LIN {X 0,Y 266.128,Z 281.314,A -85,B 0,C 180,E1 -18933.081,E2 -18933.081} C_VEL
LIN {X 0,Y 270.948,Z 292.828,A -85,B 0,C 180,E1 -18934.221,E2 -18934.221} C_VEL
LIN {X 0,Y 268.167,Z 358.472,A -85,B 0,C 180,E1 -18936.067,E2 -18936.067} C_VEL
LIN {X 0,Y 266.983,Z 371.691,A -85,B 0,C 180,E1 -18936.714,E2 -18936.714} C_VEL
LIN {X 0,Y 265.443,Z 384.254,A -85,B 0,C 180,E1 -18937.634,E2 -18937.634} C_VEL
LIN {X 0,Y 263.666,Z 395.639,A -85,B 0,C 180,E1 -18938.771,E2 -18938.771} C_VEL
LIN {X 0,Y 261.611,Z 406.363,A -85,B 0,C 180,E1 -18940.147,E2 -18940.147} C_VEL
LIN {X 0,Y 259.271,Z 416.661,A -85,B 0,C 180,E1 -18941.804,E2 -18941.804} C_VEL
LIN {X 0,Y 257.067,Z 425.49,A -85,B 0,C 180,E1 -18943.574,E2 -18943.574} C_VEL
LIN {X 0,Y 254.605,Z 434.603,A -85,B 0,C 180,E1 -18945.865,E2 -18945.865} C_VEL
LIN {X 0,Y 252.569,Z 441.662,A -85,B 0,C 180,E1 -18948.101,E2 -18948.101} C_VEL
LIN {X 0,Y 250.564,Z 448.509,A -85,B 0,C 180,E1 -18950.869,E2 -18950.869} C_VEL
LIN {X 0,Y 249.045,Z 453.666,A -85,B 0,C 180,E1 -18953.657,E2 -18953.657} C_VEL
LIN {X 0,Y 247.968,Z 457.373,A -85,B 0,C 180,E1 -18956.449,E2 -18956.449} C_VEL
LIN {X 0,Y 247.203,Z 459.794,A -85,B 0,C 180,E1 -18959.22,E2 -18959.22} C_VEL
LIN {X 0,Y 246.741,Z 461.043,A -85,B 0,C 180,E1 -18962.005,E2 -18962.005} C_VEL
LIN {X 0,Y 246.536,Z 461.149,A -85,B 0,C 180,E1 -18964.684,E2 -18964.684} C_VEL
LIN {X 0,Y 246.559,Z 460.631,A -85,B 0,C 180,E1 -18966.48,E2 -18966.48} C_VEL
LIN {X 0,Y 246.666,Z 459.608,A -85,B 0,C 180,E1 -18968.26,E2 -18968.26} C_VEL
LIN {X 0,Y 246.957,Z 458.137,A -85,B 0,C 180,E1 -18970.032,E2 -18970.032} C_VEL
LIN {X 0,Y 247.548,Z 455.004,A -85,B 0,C 180,E1 -18972.656,E2 -18972.656} C_VEL
LIN {X 0,Y 248.257,Z 450.729,A -85,B 0,C 180,E1 -18975.239,E2 -18975.239} C_VEL
LIN {X 0,Y 249.502,Z 444.093,A -85,B 0,C 180,E1 -18978.216,E2 -18978.216} C_VEL
LIN {X 0,Y 250.978,Z 436.828,A -85,B 0,C 180,E1 -18980.734,E2 -18980.734} C_VEL
LIN {X 0,Y 252.458,Z 429.359,A -85,B 0,C 180,E1 -18982.803,E2 -18982.803} C_VEL
LIN {X 0,Y 254.295,Z 419.879,A -85,B 0,C 180,E1 -18984.917,E2 -18984.917} C_VEL
LIN {X 0,Y 256.205,Z 408.995,A -85,B 0,C 180,E1 -18986.855,E2 -18986.855} C_VEL
LIN {X 0,Y 258.11,Z 397.488,A -85,B 0,C 180,E1 -18988.439,E2 -18988.439} C_VEL
LIN {X 0,Y 259.76,Z 384.646,A -85,B 0,C 180,E1 -18989.806,E2 -18989.806} C_VEL
LIN {X 0,Y 261.012,Z 371.674,A -85,B 0,C 180,E1 -18990.807,E2 -18990.807} C_VEL
LIN {X 0,Y 261.936,Z 358.441,A -85,B 0,C 180,E1 -18991.491,E2 -18991.491} C_VEL
LIN {X 0,Y 263.923,Z 304.953,A -85,B 0,C 180,E1 -18993.003,E2 -18993.003} C_VEL
LIN {X 0,Y 264.426,Z 287.5,A -85,B 0,C 180,E1 -18993.493,E2 -18993.493} C_VEL
LIN {X 0,Y 260.391,Z 275.57,A -85,B 0,C 180,E1 -18994.288,E2 -18994.288} C_VEL
LIN {X 0,Y 255.297,Z 263.136,A -85,B 0,C 180,E1 -18995.245,E2 -18995.245} C_VEL
LIN {X 0,Y 249.757,Z 250.129,A -85,B 0,C 180,E1 -18996.361,E2 -18996.361} C_VEL
LIN {X 0,Y 249.402,Z 248.419,A -85,B 0,C 180,E1 -18997.183,E2 -18997.183} C_VEL
LIN {X 0,Y 249.345,Z 248.423,A -85,B 0,C 180,E1 -18999.736,E2 -18999.736} C_VEL
LIN {X 0,Y 249.208,Z 248.445,A -85,B 0,C 180,E1 -19004.703,E2 -19004.703} C_VEL
LIN {X 0,Y 249.142,Z 248.454,A -85,B 0,C 180,E1 -19008.077,E2 -19008.077} C_VEL
LIN {X 0,Y 249.086,Z 248.455,A -85,B 0,C 180,E1 -19011.518,E2 -19011.518} C_VEL
LIN {X 0,Y 249.106,Z 248.455,A -85,B 0,C 180,E1 -19015.469,E2 -19015.469} C_VEL
LIN {X 0,Y 249.04,Z 248.456,A -85,B 0,C 180,E1 -19018.974,E2 -19018.974} C_VEL
LIN {X 0,Y 249.028,Z 248.464,A -85,B 0,C 180,E1 -19022.426,E2 -19022.426} C_VEL
LIN {X 0,Y 249.049,Z 248.456,A -85,B 0,C 180,E1 -19026.341,E2 -19026.341} C_VEL
LIN {X 0,Y 249.006,Z 248.466,A -85,B 0,C 180,E1 -19030.477,E2 -19030.477} C_VEL
LIN {X 0,Y 248.993,Z 248.458,A -85,B 0,C 180,E1 -19034.881,E2 -19034.881} C_VEL
LIN {X 0,Y 249.016,Z 248.463,A -85,B 0,C 180,E1 -19037.362,E2 -19037.362} C_VEL
LIN {X 0,Y 249.044,Z 248.454,A -85,B 0,C 180,E1 -19042.199,E2 -19042.199} C_VEL
LIN {X 0,Y 249.043,Z 248.449,A -85,B 0,C 180,E1 -19045.639,E2 -19045.639} C_VEL
LIN {X 0,Y 249.046,Z 248.46,A -85,B 0,C 180,E1 -19049.472,E2 -19049.472} C_VEL
LIN {X 0,Y 249.071,Z 248.452,A -85,B 0,C 180,E1 -19053.162,E2 -19053.162} C_VEL
LIN {X 0,Y 249.078,Z 248.441,A -85,B 0,C 180,E1 -19056.732,E2 -19056.732} C_VEL
LIN {X 0,Y 249.11,Z 248.452,A -85,B 0,C 180,E1 -19060.211,E2 -19060.211} C_VEL
LIN {X 0,Y 249.241,Z 248.437,A -85,B 0,C 180,E1 -19063.622,E2 -19063.622} C_VEL
LIN {X 0,Y 249.251,Z 248.414,A -85,B 0,C 180,E1 -19068.616,E2 -19068.616} C_VEL
LIN {X 0,Y 249.482,Z 248.398,A -85,B 0,C 180,E1 -19071.903,E2 -19071.903} C_VEL
LIN {X 0,Y 249.435,Z 248.412,A -85,B 0,C 180,E1 -19076.769,E2 -19076.769} C_VEL
LIN {X 0,Y 249.726,Z 248.366,A -85,B 0,C 180,E1 -19080,E2 -19080} C_VEL
LIN {X 0,Y 249.434,Z 248.399,A -85,B 0,C 180,E1 -19083.23,E2 -19083.23} C_VEL
LIN {X 0,Y 249.482,Z 248.409,A -85,B 0,C 180,E1 -19088.097,E2 -19088.097} C_VEL
LIN {X 0,Y 249.251,Z 248.429,A -85,B 0,C 180,E1 -19091.383,E2 -19091.383} C_VEL
LIN {X 0,Y 249.207,Z 248.425,A -85,B 0,C 180,E1 -19092.51,E2 -19092.51} C_VEL
LIN {X 0,Y 248.537,Z 248.51,A -85,B 0,C 180,E1 -19093.859,E2 -19093.859} C_VEL
LIN {X 0,Y 245.637,Z 248.881,A -85,B 0,C 180,E1 -19096.057,E2 -19096.057} C_VEL
LIN {X 0,Y 243.167,Z 249.193,A -85,B 0,C 180,E1 -19097.847,E2 -19097.847} C_VEL
LIN {X 0,Y 242.108,Z 249.325,A -85,B 0,C 180,E1 -19099.238,E2 -19099.238} C_VEL
LIN {X 0,Y 242.022,Z 249.332,A -85,B 0,C 180,E1 -19099.709,E2 -19099.709} C_VEL
LIN {X 0,Y 242.056,Z 249.329,A -85,B 0,C 180,E1 -19103.984,E2 -19103.984} C_VEL
LIN {X 0,Y 242.007,Z 249.336,A -85,B 0,C 180,E1 -19107.687,E2 -19107.687} C_VEL
LIN {X 0,Y 241.973,Z 249.342,A -85,B 0,C 180,E1 -19111.52,E2 -19111.52} C_VEL
LIN {X 0,Y 242.004,Z 249.339,A -85,B 0,C 180,E1 -19115.597,E2 -19115.597} C_VEL
LIN {X 0,Y 241.955,Z 249.345,A -85,B 0,C 180,E1 -19119.719,E2 -19119.719} C_VEL
LIN {X 0,Y 241.922,Z 249.346,A -85,B 0,C 180,E1 -19124.204,E2 -19124.204} C_VEL
LIN {X 0,Y 241.945,Z 249.35,A -85,B 0,C 180,E1 -19128.08,E2 -19128.08} C_VEL
LIN {X 0,Y 242.07,Z 249.446,A -85,B 0,C 180,E1 -19132.786,E2 -19132.786} C_VEL
LIN {X 0,Y 244.245,Z 259.241,A -85,B 0,C 180,E1 -19136.859,E2 -19136.859} C_VEL
LIN {X 0,Y 244.934,Z 262.422,A -85,B 0,C 180,E1 -19138.129,E2 -19138.129} C_VEL
LIN {X 0,Y 252.756,Z 282.367,A -85,B 0,C 180,E1 -19139.716,E2 -19139.716} C_VEL
LIN {X 0,Y 253.632,Z 285.314,A -85,B 0,C 180,E1 -19139.91,E2 -19139.91} C_VEL
LIN {X 0,Y 257.411,Z 312.087,A -85,B 0,C 180,E1 -19141.176,E2 -19141.176} C_VEL
LIN {X 0,Y 255.315,Z 370.97,A -85,B 0,C 180,E1 -19142.877,E2 -19142.877} C_VEL
LIN {X 0,Y 254.099,Z 384.714,A -85,B 0,C 180,E1 -19143.569,E2 -19143.569} C_VEL
LIN {X 0,Y 252.646,Z 397.705,A -85,B 0,C 180,E1 -19144.569,E2 -19144.569} C_VEL
LIN {X 0,Y 250.928,Z 409.521,A -85,B 0,C 180,E1 -19145.82,E2 -19145.82} C_VEL
LIN {X 0,Y 248.993,Z 420.926,A -85,B 0,C 180,E1 -19147.383,E2 -19147.383} C_VEL
LIN {X 0,Y 246.976,Z 431.203,A -85,B 0,C 180,E1 -19149.164,E2 -19149.164} C_VEL
LIN {X 0,Y 245.257,Z 440.449,A -85,B 0,C 180,E1 -19151.192,E2 -19151.192} C_VEL
LIN {X 0,Y 243.708,Z 448.08,A -85,B 0,C 180,E1 -19153.24,E2 -19153.24} C_VEL
LIN {X 0,Y 242.189,Z 455.549,A -85,B 0,C 180,E1 -19155.72,E2 -19155.72} C_VEL
LIN {X 0,Y 241.068,Z 461.533,A -85,B 0,C 180,E1 -19158.225,E2 -19158.225} C_VEL
LIN {X 0,Y 240.366,Z 466.244,A -85,B 0,C 180,E1 -19160.746,E2 -19160.746} C_VEL
LIN {X 0,Y 239.953,Z 469.818,A -85,B 0,C 180,E1 -19163.272,E2 -19163.272} C_VEL
LIN {X 0,Y 239.797,Z 471.831,A -85,B 0,C 180,E1 -19165.189,E2 -19165.189} C_VEL
LIN {X 0,Y 239.84,Z 473.941,A -85,B 0,C 180,E1 -19168.321,E2 -19168.321} C_VEL
LIN {X 0,Y 239.913,Z 474.499,A -85,B 0,C 180,E1 -19170,E2 -19170} C_VEL
LIN {X 0,Y 239.83,Z 474.623,A -85,B 0,C 180,E1 -19171.679,E2 -19171.679} C_VEL
LIN {X 0,Y 239.801,Z 473.657,A -85,B 0,C 180,E1 -19175.044,E2 -19175.044} C_VEL
LIN {X 0,Y 239.952,Z 472.594,A -85,B 0,C 180,E1 -19176.728,E2 -19176.728} C_VEL
LIN {X 0,Y 240.217,Z 471.104,A -85,B 0,C 180,E1 -19178.412,E2 -19178.412} C_VEL
LIN {X 0,Y 240.899,Z 468.07,A -85,B 0,C 180,E1 -19180.931,E2 -19180.931} C_VEL
LIN {X 0,Y 241.929,Z 463.995,A -85,B 0,C 180,E1 -19183.439,E2 -19183.439} C_VEL
LIN {X 0,Y 243.832,Z 457.761,A -85,B 0,C 180,E1 -19186.322,E2 -19186.322} C_VEL
LIN {X 0,Y 245.809,Z 450.997,A -85,B 0,C 180,E1 -19188.763,E2 -19188.763} C_VEL
LIN {X 0,Y 248.119,Z 442.786,A -85,B 0,C 180,E1 -19191.127,E2 -19191.127} C_VEL
LIN {X 0,Y 250.503,Z 434.045,A -85,B 0,C 180,E1 -19193.128,E2 -19193.128} C_VEL
LIN {X 0,Y 253.281,Z 423.502,A -85,B 0,C 180,E1 -19195.034,E2 -19195.034} C_VEL
LIN {X 0,Y 255.661,Z 413.101,A -85,B 0,C 180,E1 -19196.532,E2 -19196.532} C_VEL
LIN {X 0,Y 257.925,Z 401.697,A -85,B 0,C 180,E1 -19197.816,E2 -19197.816} C_VEL
LIN {X 0,Y 259.929,Z 388.71,A -85,B 0,C 180,E1 -19198.902,E2 -19198.902} C_VEL
LIN {X 0,Y 261.485,Z 375.958,A -85,B 0,C 180,E1 -19199.637,E2 -19199.637} C_VEL
LIN {X 0,Y 262.379,Z 362.672,A -85,B 0,C 180,E1 -19200.122,E2 -19200.122} C_VEL
LIN {X 0,Y 264.36,Z 313.239,A -85,B 0,C 180,E1 -19201.529,E2 -19201.529} C_VEL
LIN {X 0,Y 261.649,Z 294.723,A -85,B 0,C 180,E1 -19202.614,E2 -19202.614} C_VEL
LIN {X 0,Y 257.644,Z 285.16,A -85,B 0,C 180,E1 -19203.642,E2 -19203.642} C_VEL
LIN {X 0,Y 251.833,Z 273.124,A -85,B 0,C 180,E1 -19205.159,E2 -19205.159} C_VEL
LIN {X 0,Y 247.323,Z 264.812,A -85,B 0,C 180,E1 -19206.38,E2 -19206.38} C_VEL
LIN {X 0,Y 245.234,Z 260.708,A -85,B 0,C 180,E1 -19207.001,E2 -19207.001} C_VEL
LIN {X 0,Y 243.213,Z 253.602,A -85,B 0,C 180,E1 -19210.512,E2 -19210.512} C_VEL
LIN {X 0,Y 241.96,Z 249.343,A -85,B 0,C 180,E1 -19212.873,E2 -19212.873} C_VEL
LIN {X 0,Y 241.932,Z 249.352,A -85,B 0,C 180,E1 -19216.572,E2 -19216.572} C_VEL
LIN {X 0,Y 241.957,Z 249.345,A -85,B 0,C 180,E1 -19220.281,E2 -19220.281} C_VEL
LIN {X 0,Y 241.988,Z 249.334,A -85,B 0,C 180,E1 -19224.489,E2 -19224.489} C_VEL
LIN {X 0,Y 241.974,Z 249.333,A -85,B 0,C 180,E1 -19228.48,E2 -19228.48} C_VEL
LIN {X 0,Y 242.008,Z 249.329,A -85,B 0,C 180,E1 -19232.313,E2 -19232.313} C_VEL
LIN {X 0,Y 242.058,Z 249.326,A -85,B 0,C 180,E1 -19236.016,E2 -19236.016} C_VEL
LIN {X 0,Y 242.038,Z 249.335,A -85,B 0,C 180,E1 -19239.608,E2 -19239.608} C_VEL
LIN {X 0,Y 242.164,Z 249.32,A -85,B 0,C 180,E1 -19243.278,E2 -19243.278} C_VEL
LIN {X 0,Y 242.187,Z 249.316,A -85,B 0,C 180,E1 -19248.28,E2 -19248.28} C_VEL
LIN {X 0,Y 242.427,Z 249.28,A -85,B 0,C 180,E1 -19251.666,E2 -19251.666} C_VEL
LIN {X 0,Y 242.258,Z 249.296,A -85,B 0,C 180,E1 -19255.007,E2 -19255.007} C_VEL
LIN {X 0,Y 242.636,Z 249.257,A -85,B 0,C 180,E1 -19258.34,E2 -19258.34} C_VEL
LIN {X 0,Y 242.636,Z 249.261,A -85,B 0,C 180,E1 -19261.66,E2 -19261.66} C_VEL
LIN {X 0,Y 242.43,Z 249.284,A -85,B 0,C 180,E1 -19266.708,E2 -19266.708} C_VEL
LIN {X 0,Y 242.315,Z 249.302,A -85,B 0,C 180,E1 -19270.022,E2 -19270.022} C_VEL
LIN {X 0,Y 242.168,Z 249.313,A -85,B 0,C 180,E1 -19275.141,E2 -19275.141} C_VEL
LIN {X 0,Y 242.073,Z 249.326,A -85,B 0,C 180,E1 -19278.624,E2 -19278.624} C_VEL
LIN {X 0,Y 242.006,Z 249.34,A -85,B 0,C 180,E1 -19282.181,E2 -19282.181} C_VEL
LIN {X 0,Y 242.035,Z 249.495,A -85,B 0,C 180,E1 -19286.516,E2 -19286.516} C_VEL
LIN {X 0,Y 242.596,Z 251.41,A -85,B 0,C 180,E1 -19287.498,E2 -19287.498} C_VEL
LIN {X 0,Y 245.302,Z 255.739,A -85,B 0,C 180,E1 -19288.27,E2 -19288.27} C_VEL
LIN {X 0,Y 252.844,Z 268.592,A -85,B 0,C 180,E1 -19290.302,E2 -19290.302} C_VEL
LIN {X 0,Y 259.452,Z 281.589,A -85,B 0,C 180,E1 -19291.986,E2 -19291.986} C_VEL
LIN {X 0,Y 265.197,Z 295.065,A -85,B 0,C 180,E1 -19293.413,E2 -19293.413} C_VEL
LIN {X 0,Y 262.301,Z 358.088,A -85,B 0,C 180,E1 -19295.194,E2 -19295.194} C_VEL
LIN {X 0,Y 261.078,Z 371.499,A -85,B 0,C 180,E1 -19295.854,E2 -19295.854} C_VEL
LIN {X 0,Y 259.42,Z 384.584,A -85,B 0,C 180,E1 -19296.826,E2 -19296.826} C_VEL
LIN {X 0,Y 257.557,Z 395.918,A -85,B 0,C 180,E1 -19297.983,E2 -19297.983} C_VEL
LIN {X 0,Y 255.153,Z 407.642,A -85,B 0,C 180,E1 -19299.535,E2 -19299.535} C_VEL
LIN {X 0,Y 252.626,Z 418.187,A -85,B 0,C 180,E1 -19301.311,E2 -19301.311} C_VEL
LIN {X 0,Y 250.347,Z 426.756,A -85,B 0,C 180,E1 -19303.122,E2 -19303.122} C_VEL
LIN {X 0,Y 247.771,Z 435.677,A -85,B 0,C 180,E1 -19305.482,E2 -19305.482} C_VEL
LIN {X 0,Y 245.384,Z 443.543,A -85,B 0,C 180,E1 -19308.131,E2 -19308.131} C_VEL
LIN {X 0,Y 243.614,Z 449.235,A -85,B 0,C 180,E1 -19310.604,E2 -19310.604} C_VEL
LIN {X 0,Y 242.015,Z 454.238,A -85,B 0,C 180,E1 -19313.465,E2 -19313.465} C_VEL
LIN {X 0,Y 240.912,Z 457.841,A -85,B 0,C 180,E1 -19316.339,E2 -19316.339} C_VEL
LIN {X 0,Y 240.328,Z 459.538,A -85,B 0,C 180,E1 -19318.239,E2 -19318.239} C_VEL
LIN {X 0,Y 239.678,Z 461.188,A -85,B 0,C 180,E1 -19321.605,E2 -19321.605} C_VEL
LIN {X 0,Y 239.472,Z 461.423,A -85,B 0,C 180,E1 -19323.882,E2 -19323.882} C_VEL
LIN {X 0,Y 239.47,Z 461.061,A -85,B 0,C 180,E1 -19325.74,E2 -19325.74} C_VEL
LIN {X 0,Y 239.5,Z 460.259,A -85,B 0,C 180,E1 -19327.575,E2 -19327.575} C_VEL
LIN {X 0,Y 239.781,Z 458.661,A -85,B 0,C 180,E1 -19329.707,E2 -19329.707} C_VEL
LIN {X 0,Y 240.32,Z 456.053,A -85,B 0,C 180,E1 -19332.117,E2 -19332.117} C_VEL
LIN {X 0,Y 241.024,Z 452.063,A -85,B 0,C 180,E1 -19334.786,E2 -19334.786} C_VEL
LIN {X 0,Y 242,Z 446.849,A -85,B 0,C 180,E1 -19337.419,E2 -19337.419} C_VEL
LIN {X 0,Y 243.365,Z 440.237,A -85,B 0,C 180,E1 -19340.022,E2 -19340.022} C_VEL
LIN {X 0,Y 245.116,Z 431.875,A -85,B 0,C 180,E1 -19342.587,E2 -19342.587} C_VEL
LIN {X 0,Y 246.993,Z 422.758,A -85,B 0,C 180,E1 -19344.813,E2 -19344.813} C_VEL
LIN {X 0,Y 248.864,Z 412.772,A -85,B 0,C 180,E1 -19346.762,E2 -19346.762} C_VEL
LIN {X 0,Y 250.734,Z 402.199,A -85,B 0,C 180,E1 -19348.394,E2 -19348.394} C_VEL
LIN {X 0,Y 252.416,Z 390.682,A -85,B 0,C 180,E1 -19349.8,E2 -19349.8} C_VEL
LIN {X 0,Y 253.89,Z 378.372,A -85,B 0,C 180,E1 -19350.94,E2 -19350.94} C_VEL
LIN {X 0,Y 254.975,Z 365.675,A -85,B 0,C 180,E1 -19351.775,E2 -19351.775} C_VEL
LIN {X 0,Y 255.729,Z 352.726,A -85,B 0,C 180,E1 -19352.317,E2 -19352.317} C_VEL
LIN {X 0,Y 257.984,Z 288.658,A -85,B 0,C 180,E1 -19354.129,E2 -19354.129} C_VEL
LIN {X 0,Y 251.527,Z 270.992,A -85,B 0,C 180,E1 -19355.416,E2 -19355.416} C_VEL
LIN {X 0,Y 242.616,Z 250.421,A -85,B 0,C 180,E1 -19357.202,E2 -19357.202} C_VEL
LIN {X 0,Y 242.383,Z 249.294,A -85,B 0,C 180,E1 -19357.706,E2 -19357.706} C_VEL
LIN {X 0,Y 242.182,Z 249.319,A -85,B 0,C 180,E1 -19361.72,E2 -19361.72} C_VEL
LIN {X 0,Y 242.165,Z 249.323,A -85,B 0,C 180,E1 -19366.721,E2 -19366.721} C_VEL
LIN {X 0,Y 242.027,Z 249.332,A -85,B 0,C 180,E1 -19371.686,E2 -19371.686} C_VEL
LIN {X 0,Y 242.033,Z 249.338,A -85,B 0,C 180,E1 -19375.82,E2 -19375.82} C_VEL
LIN {X 0,Y 241.97,Z 249.338,A -85,B 0,C 180,E1 -19379.588,E2 -19379.588} C_VEL
LIN {X 0,Y 241.98,Z 249.343,A -85,B 0,C 180,E1 -19383.492,E2 -19383.492} C_VEL
LIN {X 0,Y 241.99,Z 249.337,A -85,B 0,C 180,E1 -19387.581,E2 -19387.581} C_VEL
LIN {X 0,Y 241.933,Z 249.343,A -85,B 0,C 180,E1 -19391.923,E2 -19391.923} C_VEL
LIN {X 0,Y 241.932,Z 249.345,A -85,B 0,C 180,E1 -19396.571,E2 -19396.571} C_VEL
LIN {X 0,Y 241.956,Z 249.343,A -85,B 0,C 180,E1 -19400.28,E2 -19400.28} C_VEL
LIN {X 0,Y 241.987,Z 249.324,A -85,B 0,C 180,E1 -19404.489,E2 -19404.489} C_VEL
LIN {X 0,Y 241.972,Z 249.342,A -85,B 0,C 180,E1 -19408.479,E2 -19408.479} C_VEL
LIN {X 0,Y 242.002,Z 249.334,A -85,B 0,C 180,E1 -19412.312,E2 -19412.312} C_VEL
LIN {X 0,Y 242.056,Z 249.312,A -85,B 0,C 180,E1 -19416.016,E2 -19416.016} C_VEL
LIN {X 0,Y 242.036,Z 249.328,A -85,B 0,C 180,E1 -19419.608,E2 -19419.608} C_VEL
LIN {X 0,Y 242.162,Z 249.318,A -85,B 0,C 180,E1 -19423.278,E2 -19423.278} C_VEL
LIN {X 0,Y 242.185,Z 249.294,A -85,B 0,C 180,E1 -19428.28,E2 -19428.28} C_VEL
LIN {X 0,Y 242.433,Z 249.274,A -85,B 0,C 180,E1 -19431.666,E2 -19431.666} C_VEL
LIN {X 0,Y 242.259,Z 249.306,A -85,B 0,C 180,E1 -19435.007,E2 -19435.007} C_VEL
LIN {X 0,Y 242.635,Z 249.255,A -85,B 0,C 180,E1 -19438.34,E2 -19438.34} C_VEL
LIN {X 0,Y 242.634,Z 249.241,A -85,B 0,C 180,E1 -19441.66,E2 -19441.66} C_VEL
LIN {X 0,Y 242.432,Z 249.286,A -85,B 0,C 180,E1 -19446.659,E2 -19446.659} C_VEL
LIN {X 0,Y 242.344,Z 249.296,A -85,B 0,C 180,E1 -19450.02,E2 -19450.02} C_VEL
LIN {X 0,Y 242.165,Z 249.31,A -85,B 0,C 180,E1 -19455.141,E2 -19455.141} C_VEL
LIN {X 0,Y 242.072,Z 249.331,A -85,B 0,C 180,E1 -19458.624,E2 -19458.624} C_VEL
LIN {X 0,Y 242.022,Z 249.332,A -85,B 0,C 180,E1 -19459.709,E2 -19459.709} C_VEL
LIN {X 0,Y 241.363,Z 249.417,A -85,B 0,C 180,E1 -19461.098,E2 -19461.098} C_VEL
LIN {X 0,Y 238.532,Z 249.775,A -85,B 0,C 180,E1 -19463.364,E2 -19463.364} C_VEL
LIN {X 0,Y 236.107,Z 250.077,A -85,B 0,C 180,E1 -19465.209,E2 -19465.209} C_VEL
LIN {X 0,Y 235.04,Z 250.206,A -85,B 0,C 180,E1 -19466.641,E2 -19466.641} C_VEL
LIN {X 0,Y 234.939,Z 250.214,A -85,B 0,C 180,E1 -19467.127,E2 -19467.127} C_VEL
LIN {X 0,Y 234.93,Z 250.222,A -85,B 0,C 180,E1 -19470.568,E2 -19470.568} C_VEL
LIN {X 0,Y 234.929,Z 250.221,A -85,B 0,C 180,E1 -19474.638,E2 -19474.638} C_VEL
LIN {X 0,Y 234.94,Z 250.219,A -85,B 0,C 180,E1 -19478.945,E2 -19478.945} C_VEL
LIN {X 0,Y 234.879,Z 250.219,A -85,B 0,C 180,E1 -19483.488,E2 -19483.488} C_VEL
LIN {X 0,Y 234.886,Z 250.227,A -85,B 0,C 180,E1 -19486.514,E2 -19486.514} C_VEL
LIN {X 0,Y 234.954,Z 250.212,A -85,B 0,C 180,E1 -19491.086,E2 -19491.086} C_VEL
LIN {X 0,Y 235.002,Z 250.334,A -85,B 0,C 180,E1 -19492.121,E2 -19492.121} C_VEL
LIN {X 0,Y 237.1,Z 259.527,A -85,B 0,C 180,E1 -19496.095,E2 -19496.095} C_VEL
LIN {X 0,Y 237.716,Z 262.328,A -85,B 0,C 180,E1 -19497.215,E2 -19497.215} C_VEL
LIN {X 0,Y 245.795,Z 282.465,A -85,B 0,C 180,E1 -19498.919,E2 -19498.919} C_VEL
LIN {X 0,Y 247.395,Z 287.334,A -85,B 0,C 180,E1 -19499.272,E2 -19499.272} C_VEL
LIN {X 0,Y 250.943,Z 313.525,A -85,B 0,C 180,E1 -19500.542,E2 -19500.542} C_VEL
LIN {X 0,Y 248.759,Z 371.621,A -85,B 0,C 180,E1 -19502.272,E2 -19502.272} C_VEL
LIN {X 0,Y 247.494,Z 385.083,A -85,B 0,C 180,E1 -19502.978,E2 -19502.978} C_VEL
LIN {X 0,Y 246.095,Z 397.387,A -85,B 0,C 180,E1 -19503.955,E2 -19503.955} C_VEL
LIN {X 0,Y 244.453,Z 408.44,A -85,B 0,C 180,E1 -19505.136,E2 -19505.136} C_VEL
LIN {X 0,Y 242.432,Z 420.007,A -85,B 0,C 180,E1 -19506.736,E2 -19506.736} C_VEL
LIN {X 0,Y 240.331,Z 430.432,A -85,B 0,C 180,E1 -19508.56,E2 -19508.56} C_VEL
LIN {X 0,Y 238.299,Z 440.691,A -85,B 0,C 180,E1 -19510.863,E2 -19510.863} C_VEL
LIN {X 0,Y 236.893,Z 447.513,A -85,B 0,C 180,E1 -19512.742,E2 -19512.742} C_VEL
LIN {X 0,Y 235.295,Z 455.05,A -85,B 0,C 180,E1 -19515.293,E2 -19515.293} C_VEL
LIN {X 0,Y 234.061,Z 461.09,A -85,B 0,C 180,E1 -19517.867,E2 -19517.867} C_VEL
LIN {X 0,Y 233.314,Z 465.856,A -85,B 0,C 180,E1 -19520.464,E2 -19520.464} C_VEL
LIN {X 0,Y 232.888,Z 469.48,A -85,B 0,C 180,E1 -19523.067,E2 -19523.067} C_VEL
LIN {X 0,Y 232.715,Z 471.736,A -85,B 0,C 180,E1 -19525.277,E2 -19525.277} C_VEL
LIN {X 0,Y 232.752,Z 473.691,A -85,B 0,C 180,E1 -19528.27,E2 -19528.27} C_VEL
LIN {X 0,Y 232.822,Z 474.269,A -85,B 0,C 180,E1 -19530,E2 -19530} C_VEL
LIN {X 0,Y 232.742,Z 474.435,A -85,B 0,C 180,E1 -19531.731,E2 -19531.731} C_VEL
LIN {X 0,Y 232.731,Z 473.513,A -85,B 0,C 180,E1 -19535.198,E2 -19535.198} C_VEL
LIN {X 0,Y 232.89,Z 472.471,A -85,B 0,C 180,E1 -19536.933,E2 -19536.933} C_VEL
LIN {X 0,Y 233.186,Z 471.023,A -85,B 0,C 180,E1 -19538.667,E2 -19538.667} C_VEL
LIN {X 0,Y 233.914,Z 468.025,A -85,B 0,C 180,E1 -19541.262,E2 -19541.262} C_VEL
LIN {X 0,Y 234.997,Z 463.995,A -85,B 0,C 180,E1 -19543.843,E2 -19543.843} C_VEL
LIN {X 0,Y 237.028,Z 457.826,A -85,B 0,C 180,E1 -19546.804,E2 -19546.804} C_VEL
LIN {X 0,Y 239.431,Z 450.096,A -85,B 0,C 180,E1 -19549.656,E2 -19549.656} C_VEL
LIN {X 0,Y 241.509,Z 443.011,A -85,B 0,C 180,E1 -19551.734,E2 -19551.734} C_VEL
LIN {X 0,Y 244.01,Z 434.411,A -85,B 0,C 180,E1 -19553.78,E2 -19553.78} C_VEL
LIN {X 0,Y 246.902,Z 423.998,A -85,B 0,C 180,E1 -19555.727,E2 -19555.727} C_VEL
LIN {X 0,Y 249.372,Z 413.743,A -85,B 0,C 180,E1 -19557.256,E2 -19557.256} C_VEL
LIN {X 0,Y 251.714,Z 402.56,A -85,B 0,C 180,E1 -19558.564,E2 -19558.564} C_VEL
LIN {X 0,Y 253.793,Z 390.029,A -85,B 0,C 180,E1 -19559.669,E2 -19559.669} C_VEL
LIN {X 0,Y 255.483,Z 376.775,A -85,B 0,C 180,E1 -19560.477,E2 -19560.477} C_VEL
LIN {X 0,Y 256.48,Z 363.996,A -85,B 0,C 180,E1 -19560.973,E2 -19560.973} C_VEL
LIN {X 0,Y 258.585,Z 314.433,A -85,B 0,C 180,E1 -19562.41,E2 -19562.41} C_VEL
LIN {X 0,Y 256.155,Z 297.133,A -85,B 0,C 180,E1 -19563.459,E2 -19563.459} C_VEL
LIN {X 0,Y 249.704,Z 282.43,A -85,B 0,C 180,E1 -19565.205,E2 -19565.205} C_VEL
LIN {X 0,Y 243.232,Z 269.908,A -85,B 0,C 180,E1 -19567.029,E2 -19567.029} C_VEL
LIN {X 0,Y 239.919,Z 264.16,A -85,B 0,C 180,E1 -19568.002,E2 -19568.002} C_VEL
LIN {X 0,Y 237.878,Z 260.328,A -85,B 0,C 180,E1 -19568.689,E2 -19568.689} C_VEL
LIN {X 0,Y 235.649,Z 252.613,A -85,B 0,C 180,E1 -19572.815,E2 -19572.815} C_VEL
LIN {X 0,Y 234.88,Z 250.228,A -85,B 0,C 180,E1 -19574.224,E2 -19574.224} C_VEL
LIN {X 0,Y 234.883,Z 250.223,A -85,B 0,C 180,E1 -19578.832,E2 -19578.832} C_VEL
LIN {X 0,Y 234.918,Z 250.216,A -85,B 0,C 180,E1 -19581.079,E2 -19581.079} C_VEL
LIN {X 0,Y 234.931,Z 250.212,A -85,B 0,C 180,E1 -19585.362,E2 -19585.362} C_VEL
LIN {X 0,Y 234.932,Z 250.212,A -85,B 0,C 180,E1 -19589.432,E2 -19589.432} C_VEL
LIN {X 0,Y 234.995,Z 250.207,A -85,B 0,C 180,E1 -19593.794,E2 -19593.794} C_VEL
LIN {X 0,Y 235.012,Z 250.212,A -85,B 0,C 180,E1 -19598.97,E2 -19598.97} C_VEL
LIN {X 0,Y 235.097,Z 250.197,A -85,B 0,C 180,E1 -19603.059,E2 -19603.059} C_VEL
LIN {X 0,Y 235.147,Z 250.193,A -85,B 0,C 180,E1 -19607.924,E2 -19607.924} C_VEL
LIN {X 0,Y 235.376,Z 250.155,A -85,B 0,C 180,E1 -19611.414,E2 -19611.414} C_VEL
LIN {X 0,Y 235.403,Z 250.161,A -85,B 0,C 180,E1 -19613.141,E2 -19613.141} C_VEL
LIN {X 0,Y 235.596,Z 250.134,A -85,B 0,C 180,E1 -19618.291,E2 -19618.291} C_VEL
LIN {X 0,Y 235.596,Z 250.138,A -85,B 0,C 180,E1 -19621.71,E2 -19621.71} C_VEL
LIN {X 0,Y 235.404,Z 250.158,A -85,B 0,C 180,E1 -19626.859,E2 -19626.859} C_VEL
LIN {X 0,Y 235.239,Z 250.183,A -85,B 0,C 180,E1 -19630.327,E2 -19630.327} C_VEL
LIN {X 0,Y 235.115,Z 250.192,A -85,B 0,C 180,E1 -19635.607,E2 -19635.607} C_VEL
LIN {X 0,Y 235.009,Z 250.209,A -85,B 0,C 180,E1 -19639.206,E2 -19639.206} C_VEL
LIN {X 0,Y 234.951,Z 250.219,A -85,B 0,C 180,E1 -19642.884,E2 -19642.884} C_VEL
LIN {X 0,Y 234.981,Z 250.31,A -85,B 0,C 180,E1 -19645.071,E2 -19645.071} C_VEL
LIN {X 0,Y 235.378,Z 251.736,A -85,B 0,C 180,E1 -19645.82,E2 -19645.82} C_VEL
LIN {X 0,Y 237.58,Z 255.347,A -85,B 0,C 180,E1 -19646.519,E2 -19646.519} C_VEL
LIN {X 0,Y 239.548,Z 258.341,A -85,B 0,C 180,E1 -19647.108,E2 -19647.108} C_VEL
LIN {X 0,Y 246.236,Z 269.361,A -85,B 0,C 180,E1 -19649.026,E2 -19649.026} C_VEL
LIN {X 0,Y 253.083,Z 282.429,A -85,B 0,C 180,E1 -19650.877,E2 -19650.877} C_VEL
LIN {X 0,Y 259.209,Z 296.474,A -85,B 0,C 180,E1 -19652.49,E2 -19652.49} C_VEL
LIN {X 0,Y 259.342,Z 298.411,A -85,B 0,C 180,E1 -19652.583,E2 -19652.583} C_VEL
LIN {X 0,Y 256.343,Z 359.418,A -85,B 0,C 180,E1 -19654.35,E2 -19654.35} C_VEL
LIN {X 0,Y 255.027,Z 373.007,A -85,B 0,C 180,E1 -19655.057,E2 -19655.057} C_VEL
LIN {X 0,Y 253.367,Z 385.354,A -85,B 0,C 180,E1 -19656.017,E2 -19656.017} C_VEL
LIN {X 0,Y 251.426,Z 396.504,A -85,B 0,C 180,E1 -19657.189,E2 -19657.189} C_VEL
LIN {X 0,Y 248.958,Z 408.041,A -85,B 0,C 180,E1 -19658.754,E2 -19658.754} C_VEL
LIN {X 0,Y 246.251,Z 418.766,A -85,B 0,C 180,E1 -19660.608,E2 -19660.608} C_VEL
LIN {X 0,Y 243.636,Z 428.009,A -85,B 0,C 180,E1 -19662.644,E2 -19662.644} C_VEL
LIN {X 0,Y 240.979,Z 436.765,A -85,B 0,C 180,E1 -19665.074,E2 -19665.074} C_VEL
LIN {X 0,Y 238.811,Z 443.431,A -85,B 0,C 180,E1 -19667.401,E2 -19667.401} C_VEL
LIN {X 0,Y 236.833,Z 449.403,A -85,B 0,C 180,E1 -19670.045,E2 -19670.045} C_VEL
LIN {X 0,Y 235.454,Z 453.353,A -85,B 0,C 180,E1 -19672.273,E2 -19672.273} C_VEL
LIN {X 0,Y 234.173,Z 457.304,A -85,B 0,C 180,E1 -19675.234,E2 -19675.234} C_VEL
LIN {X 0,Y 233.451,Z 459.372,A -85,B 0,C 180,E1 -19677.452,E2 -19677.452} C_VEL
LIN {X 0,Y 232.993,Z 460.521,A -85,B 0,C 180,E1 -19679.15,E2 -19679.15} C_VEL
LIN {X 0,Y 232.644,Z 461.333,A -85,B 0,C 180,E1 -19681.172,E2 -19681.172} C_VEL
LIN {X 0,Y 232.426,Z 461.63,A -85,B 0,C 180,E1 -19683.027,E2 -19683.027} C_VEL
LIN {X 0,Y 232.352,Z 461.404,A -85,B 0,C 180,E1 -19685.152,E2 -19685.152} C_VEL
LIN {X 0,Y 232.363,Z 460.788,A -85,B 0,C 180,E1 -19686.846,E2 -19686.846} C_VEL
LIN {X 0,Y 232.672,Z 459.096,A -85,B 0,C 180,E1 -19689.452,E2 -19689.452} C_VEL
LIN {X 0,Y 233.305,Z 455.934,A -85,B 0,C 180,E1 -19692.468,E2 -19692.468} C_VEL
LIN {X 0,Y 234.039,Z 451.844,A -85,B 0,C 180,E1 -19695.212,E2 -19695.212} C_VEL
LIN {X 0,Y 235.099,Z 446.516,A -85,B 0,C 180,E1 -19697.921,E2 -19697.921} C_VEL
LIN {X 0,Y 236.564,Z 439.723,A -85,B 0,C 180,E1 -19700.596,E2 -19700.596} C_VEL
LIN {X 0,Y 238.424,Z 431.205,A -85,B 0,C 180,E1 -19703.228,E2 -19703.228} C_VEL
LIN {X 0,Y 240.291,Z 422.458,A -85,B 0,C 180,E1 -19705.386,E2 -19705.386} C_VEL
LIN {X 0,Y 242.145,Z 412.834,A -85,B 0,C 180,E1 -19707.296,E2 -19707.296} C_VEL
LIN {X 0,Y 244.085,Z 402.231,A -85,B 0,C 180,E1 -19708.969,E2 -19708.969} C_VEL
LIN {X 0,Y 245.83,Z 390.664,A -85,B 0,C 180,E1 -19710.411,E2 -19710.411} C_VEL
LIN {X 0,Y 247.236,Z 379.371,A -85,B 0,C 180,E1 -19711.489,E2 -19711.489} C_VEL
LIN {X 0,Y 248.361,Z 367.271,A -85,B 0,C 180,E1 -19712.331,E2 -19712.331} C_VEL
LIN {X 0,Y 249.157,Z 353.963,A -85,B 0,C 180,E1 -19712.93,E2 -19712.93} C_VEL
LIN {X 0,Y 251.626,Z 290.598,A -85,B 0,C 180,E1 -19714.755,E2 -19714.755} C_VEL
LIN {X 0,Y 245.646,Z 274.036,A -85,B 0,C 180,E1 -19716.004,E2 -19716.004} C_VEL
LIN {X 0,Y 236.224,Z 252.784,A -85,B 0,C 180,E1 -19717.934,E2 -19717.934} C_VEL
LIN {X 0,Y 235.433,Z 250.591,A -85,B 0,C 180,E1 -19718.152,E2 -19718.152} C_VEL
LIN {X 0,Y 235.338,Z 250.174,A -85,B 0,C 180,E1 -19718.371,E2 -19718.371} C_VEL
LIN {X 0,Y 235.116,Z 250.199,A -85,B 0,C 180,E1 -19722.078,E2 -19722.078} C_VEL
LIN {X 0,Y 235.099,Z 250.204,A -85,B 0,C 180,E1 -19726.94,E2 -19726.94} C_VEL
LIN {X 0,Y 234.99,Z 250.205,A -85,B 0,C 180,E1 -19732.006,E2 -19732.006} C_VEL
LIN {X 0,Y 234.947,Z 250.216,A -85,B 0,C 180,E1 -19736.66,E2 -19736.66} C_VEL
LIN {X 0,Y 234.9,Z 250.224,A -85,B 0,C 180,E1 -19740.572,E2 -19740.572} C_VEL
LIN {X 0,Y 234.931,Z 250.212,A -85,B 0,C 180,E1 -19744.637,E2 -19744.637} C_VEL
LIN {X 0,Y 234.942,Z 250.218,A -85,B 0,C 180,E1 -19748.944,E2 -19748.944} C_VEL
LIN {X 0,Y 234.88,Z 250.215,A -85,B 0,C 180,E1 -19753.487,E2 -19753.487} C_VEL
LIN {X 0,Y 234.885,Z 250.223,A -85,B 0,C 180,E1 -19756.513,E2 -19756.513} C_VEL
LIN {X 0,Y 234.918,Z 250.218,A -85,B 0,C 180,E1 -19761.078,E2 -19761.078} C_VEL
LIN {X 0,Y 234.93,Z 250.203,A -85,B 0,C 180,E1 -19765.362,E2 -19765.362} C_VEL
LIN {X 0,Y 234.921,Z 250.22,A -85,B 0,C 180,E1 -19769.43,E2 -19769.43} C_VEL
LIN {X 0,Y 234.993,Z 250.201,A -85,B 0,C 180,E1 -19773.794,E2 -19773.794} C_VEL
LIN {X 0,Y 235.01,Z 250.202,A -85,B 0,C 180,E1 -19778.97,E2 -19778.97} C_VEL
LIN {X 0,Y 235.095,Z 250.198,A -85,B 0,C 180,E1 -19783.059,E2 -19783.059} C_VEL
LIN {X 0,Y 235.145,Z 250.172,A -85,B 0,C 180,E1 -19787.923,E2 -19787.923} C_VEL
LIN {X 0,Y 235.389,Z 250.15,A -85,B 0,C 180,E1 -19791.414,E2 -19791.414} C_VEL
LIN {X 0,Y 235.404,Z 250.156,A -85,B 0,C 180,E1 -19793.141,E2 -19793.141} C_VEL
LIN {X 0,Y 235.595,Z 250.132,A -85,B 0,C 180,E1 -19798.29,E2 -19798.29} C_VEL
LIN {X 0,Y 235.594,Z 250.116,A -85,B 0,C 180,E1 -19801.709,E2 -19801.709} C_VEL
LIN {X 0,Y 235.404,Z 250.16,A -85,B 0,C 180,E1 -19806.859,E2 -19806.859} C_VEL
LIN {X 0,Y 235.252,Z 250.176,A -85,B 0,C 180,E1 -19810.326,E2 -19810.326} C_VEL
LIN {X 0,Y 235.112,Z 250.189,A -85,B 0,C 180,E1 -19815.606,E2 -19815.606} C_VEL
LIN {X 0,Y 234.985,Z 250.208,A -85,B 0,C 180,E1 -19819.698,E2 -19819.698} C_VEL
LIN {X 0,Y 234.96,Z 250.211,A -85,B 0,C 180,E1 -19822.883,E2 -19822.883} C_VEL
LIN {X 0,Y 234.939,Z 250.214,A -85,B 0,C 180,E1 -19827.127,E2 -19827.127} C_VEL
LIN {X 0,Y 234.231,Z 250.303,A -85,B 0,C 180,E1 -19828.557,E2 -19828.557} C_VEL
LIN {X 0,Y 231.358,Z 250.666,A -85,B 0,C 180,E1 -19830.89,E2 -19830.89} C_VEL
LIN {X 0,Y 228.945,Z 250.962,A -85,B 0,C 180,E1 -19832.793,E2 -19832.793} C_VEL
LIN {X 0,Y 227.918,Z 251.091,A -85,B 0,C 180,E1 -19834.27,E2 -19834.27} C_VEL
LIN {X 0,Y 227.837,Z 251.097,A -85,B 0,C 180,E1 -19834.77,E2 -19834.77} C_VEL
LIN {X 0,Y 227.843,Z 251.101,A -85,B 0,C 180,E1 -19838.091,E2 -19838.091} C_VEL
LIN {X 0,Y 227.805,Z 251.097,A -85,B 0,C 180,E1 -19842.744,E2 -19842.744} C_VEL
LIN {X 0,Y 227.814,Z 251.108,A -85,B 0,C 180,E1 -19847.259,E2 -19847.259} C_VEL
LIN {X 0,Y 227.929,Z 251.16,A -85,B 0,C 180,E1 -19851.393,E2 -19851.393} C_VEL
LIN {X 0,Y 230.095,Z 260.44,A -85,B 0,C 180,E1 -19855.557,E2 -19855.557} C_VEL
LIN {X 0,Y 230.381,Z 261.986,A -85,B 0,C 180,E1 -19856.217,E2 -19856.217} C_VEL
LIN {X 0,Y 238.924,Z 282.85,A -85,B 0,C 180,E1 -19858.095,E2 -19858.095} C_VEL
LIN {X 0,Y 241.146,Z 288.89,A -85,B 0,C 180,E1 -19858.581,E2 -19858.581} C_VEL
LIN {X 0,Y 244.539,Z 313.529,A -85,B 0,C 180,E1 -19859.83,E2 -19859.83} C_VEL
LIN {X 0,Y 242.276,Z 371.138,A -85,B 0,C 180,E1 -19861.582,E2 -19861.582} C_VEL
LIN {X 0,Y 241.026,Z 384.704,A -85,B 0,C 180,E1 -19862.309,E2 -19862.309} C_VEL
LIN {X 0,Y 239.574,Z 397.065,A -85,B 0,C 180,E1 -19863.308,E2 -19863.308} C_VEL
LIN {X 0,Y 237.994,Z 407.342,A -85,B 0,C 180,E1 -19864.414,E2 -19864.414} C_VEL
LIN {X 0,Y 235.813,Z 419.07,A -85,B 0,C 180,E1 -19866.042,E2 -19866.042} C_VEL
LIN {X 0,Y 233.665,Z 429.627,A -85,B 0,C 180,E1 -19867.916,E2 -19867.916} C_VEL
LIN {X 0,Y 231.71,Z 439.315,A -85,B 0,C 180,E1 -19870.096,E2 -19870.096} C_VEL
LIN {X 0,Y 230.105,Z 446.936,A -85,B 0,C 180,E1 -19872.217,E2 -19872.217} C_VEL
LIN {X 0,Y 228.405,Z 454.54,A -85,B 0,C 180,E1 -19874.839,E2 -19874.839} C_VEL
LIN {X 0,Y 227.069,Z 460.639,A -85,B 0,C 180,E1 -19877.488,E2 -19877.488} C_VEL
LIN {X 0,Y 226.285,Z 465.46,A -85,B 0,C 180,E1 -19880.165,E2 -19880.165} C_VEL
LIN {X 0,Y 225.819,Z 469.135,A -85,B 0,C 180,E1 -19882.849,E2 -19882.849} C_VEL
LIN {X 0,Y 225.608,Z 471.699,A -85,B 0,C 180,E1 -19885.447,E2 -19885.447} C_VEL
LIN {X 0,Y 225.666,Z 473.439,A -85,B 0,C 180,E1 -19888.216,E2 -19888.216} C_VEL
LIN {X 0,Y 225.734,Z 474.039,A -85,B 0,C 180,E1 -19890,E2 -19890} C_VEL
LIN {X 0,Y 225.655,Z 474.238,A -85,B 0,C 180,E1 -19891.785,E2 -19891.785} C_VEL
LIN {X 0,Y 225.596,Z 473.729,A -85,B 0,C 180,E1 -19894.513,E2 -19894.513} C_VEL
LIN {X 0,Y 225.822,Z 472.348,A -85,B 0,C 180,E1 -19897.151,E2 -19897.151} C_VEL
LIN {X 0,Y 226.143,Z 470.932,A -85,B 0,C 180,E1 -19898.94,E2 -19898.94} C_VEL
LIN {X 0,Y 226.946,Z 467.975,A -85,B 0,C 180,E1 -19901.613,E2 -19901.613} C_VEL
LIN {X 0,Y 228.079,Z 464.001,A -85,B 0,C 180,E1 -19904.271,E2 -19904.271} C_VEL
LIN {X 0,Y 229.882,Z 458.909,A -85,B 0,C 180,E1 -19906.884,E2 -19906.884} C_VEL
LIN {X 0,Y 231.99,Z 452.537,A -85,B 0,C 180,E1 -19909.466,E2 -19909.466} C_VEL
LIN {X 0,Y 234.432,Z 444.892,A -85,B 0,C 180,E1 -19911.916,E2 -19911.916} C_VEL
LIN {X 0,Y 236.991,Z 436.534,A -85,B 0,C 180,E1 -19914.064,E2 -19914.064} C_VEL
LIN {X 0,Y 239.905,Z 426.725,A -85,B 0,C 180,E1 -19916.067,E2 -19916.067} C_VEL
LIN {X 0,Y 242.793,Z 415.8,A -85,B 0,C 180,E1 -19917.824,E2 -19917.824} C_VEL
LIN {X 0,Y 245.183,Z 405.149,A -85,B 0,C 180,E1 -19919.163,E2 -19919.163} C_VEL
LIN {X 0,Y 247.518,Z 392.434,A -85,B 0,C 180,E1 -19920.382,E2 -19920.382} C_VEL
LIN {X 0,Y 249.347,Z 379.665,A -85,B 0,C 180,E1 -19921.251,E2 -19921.251} C_VEL
LIN {X 0,Y 250.572,Z 365.985,A -85,B 0,C 180,E1 -19921.847,E2 -19921.847} C_VEL
LIN {X 0,Y 252.907,Z 315.542,A -85,B 0,C 180,E1 -19923.342,E2 -19923.342} C_VEL
LIN {X 0,Y 250.842,Z 300.132,A -85,B 0,C 180,E1 -19924.304,E2 -19924.304} C_VEL
LIN {X 0,Y 244.74,Z 286.055,A -85,B 0,C 180,E1 -19926.046,E2 -19926.046} C_VEL
LIN {X 0,Y 238.658,Z 274.16,A -85,B 0,C 180,E1 -19927.855,E2 -19927.855} C_VEL
LIN {X 0,Y 233.56,Z 265.175,A -85,B 0,C 180,E1 -19929.461,E2 -19929.461} C_VEL
LIN {X 0,Y 230.836,Z 260.821,A -85,B 0,C 180,E1 -19930.36,E2 -19930.36} C_VEL
LIN {X 0,Y 230.519,Z 260.07,A -85,B 0,C 180,E1 -19930.51,E2 -19930.51} C_VEL
LIN {X 0,Y 228.8,Z 254.331,A -85,B 0,C 180,E1 -19933.793,E2 -19933.793} C_VEL
LIN {X 0,Y 227.844,Z 251.102,A -85,B 0,C 180,E1 -19935.768,E2 -19935.768} C_VEL
LIN {X 0,Y 227.853,Z 251.099,A -85,B 0,C 180,E1 -19940.454,E2 -19940.454} C_VEL
LIN {X 0,Y 227.881,Z 251.092,A -85,B 0,C 180,E1 -19944.128,E2 -19944.128} C_VEL
LIN {X 0,Y 227.871,Z 251.089,A -85,B 0,C 180,E1 -19948.378,E2 -19948.378} C_VEL
LIN {X 0,Y 227.887,Z 251.087,A -85,B 0,C 180,E1 -19952.445,E2 -19952.445} C_VEL
LIN {X 0,Y 227.915,Z 251.085,A -85,B 0,C 180,E1 -19956.368,E2 -19956.368} C_VEL
LIN {X 0,Y 227.943,Z 251.086,A -85,B 0,C 180,E1 -19960.175,E2 -19960.175} C_VEL
LIN {X 0,Y 228.058,Z 251.076,A -85,B 0,C 180,E1 -19963.898,E2 -19963.898} C_VEL
LIN {X 0,Y 228.094,Z 251.068,A -85,B 0,C 180,E1 -19967.545,E2 -19967.545} C_VEL
LIN {X 0,Y 228.306,Z 251.034,A -85,B 0,C 180,E1 -19971.146,E2 -19971.146} C_VEL
LIN {X 0,Y 228.354,Z 251.041,A -85,B 0,C 180,E1 -19972.929,E2 -19972.929} C_VEL
LIN {X 0,Y 228.555,Z 251.012,A -85,B 0,C 180,E1 -19978.238,E2 -19978.238} C_VEL
LIN {X 0,Y 228.555,Z 251.016,A -85,B 0,C 180,E1 -19981.762,E2 -19981.762} C_VEL
LIN {X 0,Y 228.355,Z 251.034,A -85,B 0,C 180,E1 -19987.072,E2 -19987.072} C_VEL
LIN {X 0,Y 228.16,Z 251.061,A -85,B 0,C 180,E1 -19990.651,E2 -19990.651} C_VEL
LIN {X 0,Y 228.066,Z 251.073,A -85,B 0,C 180,E1 -19994.272,E2 -19994.272} C_VEL
LIN {X 0,Y 228.004,Z 251.079,A -85,B 0,C 180,E1 -19997.953,E2 -19997.953} C_VEL
LIN {X 0,Y 227.929,Z 251.094,A -85,B 0,C 180,E1 -20002.803,E2 -20002.803} C_VEL
LIN {X 0,Y 227.911,Z 251.252,A -85,B 0,C 180,E1 -20003.529,E2 -20003.529} C_VEL
LIN {X 0,Y 228.072,Z 251.981,A -85,B 0,C 180,E1 -20003.917,E2 -20003.917} C_VEL
LIN {X 0,Y 229.31,Z 254.542,A -85,B 0,C 180,E1 -20004.381,E2 -20004.381} C_VEL
LIN {X 0,Y 231.515,Z 257.125,A -85,B 0,C 180,E1 -20005.09,E2 -20005.09} C_VEL
LIN {X 0,Y 237.4,Z 266.36,A -85,B 0,C 180,E1 -20006.964,E2 -20006.964} C_VEL
LIN {X 0,Y 244.019,Z 277.987,A -85,B 0,C 180,E1 -20008.917,E2 -20008.917} C_VEL
LIN {X 0,Y 250.153,Z 290.635,A -85,B 0,C 180,E1 -20010.646,E2 -20010.646} C_VEL
LIN {X 0,Y 253.685,Z 298.942,A -85,B 0,C 180,E1 -20011.614,E2 -20011.614} C_VEL
LIN {X 0,Y 250.633,Z 359.231,A -85,B 0,C 180,E1 -20013.4,E2 -20013.4} C_VEL
LIN {X 0,Y 249.309,Z 372.596,A -85,B 0,C 180,E1 -20014.099,E2 -20014.099} C_VEL
LIN {X 0,Y 247.5,Z 385.416,A -85,B 0,C 180,E1 -20015.099,E2 -20015.099} C_VEL
LIN {X 0,Y 245.377,Z 396.965,A -85,B 0,C 180,E1 -20016.337,E2 -20016.337} C_VEL
LIN {X 0,Y 242.684,Z 409.015,A -85,B 0,C 180,E1 -20018.023,E2 -20018.023} C_VEL
LIN {X 0,Y 240.065,Z 418.908,A -85,B 0,C 180,E1 -20019.784,E2 -20019.784} C_VEL
LIN {X 0,Y 237.554,Z 427.401,A -85,B 0,C 180,E1 -20021.667,E2 -20021.667} C_VEL
LIN {X 0,Y 234.734,Z 436.049,A -85,B 0,C 180,E1 -20024.064,E2 -20024.064} C_VEL
LIN {X 0,Y 232.396,Z 443.094,A -85,B 0,C 180,E1 -20026.535,E2 -20026.535} C_VEL
LIN {X 0,Y 230.389,Z 448.722,A -85,B 0,C 180,E1 -20029.017,E2 -20029.017} C_VEL
LIN {X 0,Y 228.474,Z 453.99,A -85,B 0,C 180,E1 -20032.033,E2 -20032.033} C_VEL
LIN {X 0,Y 227.128,Z 457.779,A -85,B 0,C 180,E1 -20035.079,E2 -20035.079} C_VEL
LIN {X 0,Y 226.157,Z 460.272,A -85,B 0,C 180,E1 -20038.11,E2 -20038.11} C_VEL
LIN {X 0,Y 225.594,Z 461.482,A -85,B 0,C 180,E1 -20040.727,E2 -20040.727} C_VEL
LIN {X 0,Y 225.263,Z 461.767,A -85,B 0,C 180,E1 -20044.101,E2 -20044.101} C_VEL
LIN {X 0,Y 225.245,Z 461.306,A -85,B 0,C 180,E1 -20046.07,E2 -20046.07} C_VEL
LIN {X 0,Y 225.516,Z 459.504,A -85,B 0,C 180,E1 -20049.216,E2 -20049.216} C_VEL
LIN {X 0,Y 226.301,Z 455.813,A -85,B 0,C 180,E1 -20052.84,E2 -20052.84} C_VEL
LIN {X 0,Y 227.08,Z 451.621,A -85,B 0,C 180,E1 -20055.665,E2 -20055.665} C_VEL
LIN {X 0,Y 228.216,Z 446.15,A -85,B 0,C 180,E1 -20058.453,E2 -20058.453} C_VEL
LIN {X 0,Y 229.779,Z 439.203,A -85,B 0,C 180,E1 -20061.203,E2 -20061.203} C_VEL
LIN {X 0,Y 231.755,Z 430.536,A -85,B 0,C 180,E1 -20063.907,E2 -20063.907} C_VEL
LIN {X 0,Y 233.766,Z 421.32,A -85,B 0,C 180,E1 -20066.171,E2 -20066.171} C_VEL
LIN {X 0,Y 235.911,Z 410.453,A -85,B 0,C 180,E1 -20068.293,E2 -20068.293} C_VEL
LIN {X 0,Y 237.987,Z 399.251,A -85,B 0,C 180,E1 -20070,E2 -20070} C_VEL
LIN {X 0,Y 239.71,Z 387.936,A -85,B 0,C 180,E1 -20071.337,E2 -20071.337} C_VEL
LIN {X 0,Y 241.15,Z 374.906,A -85,B 0,C 180,E1 -20072.505,E2 -20072.505} C_VEL
LIN {X 0,Y 242.257,Z 362.335,A -85,B 0,C 180,E1 -20073.274,E2 -20073.274} C_VEL
LIN {X 0,Y 243.052,Z 346.977,A -85,B 0,C 180,E1 -20073.825,E2 -20073.825} C_VEL
LIN {X 0,Y 245.197,Z 291.869,A -85,B 0,C 180,E1 -20075.448,E2 -20075.448} C_VEL
LIN {X 0,Y 239.128,Z 275.515,A -85,B 0,C 180,E1 -20076.751,E2 -20076.751} C_VEL
LIN {X 0,Y 229.976,Z 254.858,A -85,B 0,C 180,E1 -20078.716,E2 -20078.716} C_VEL
LIN {X 0,Y 228.479,Z 252.089,A -85,B 0,C 180,E1 -20079.033,E2 -20079.033} C_VEL
LIN {X 0,Y 228.249,Z 251.052,A -85,B 0,C 180,E1 -20079.125,E2 -20079.125} C_VEL
LIN {X 0,Y 228.067,Z 251.08,A -85,B 0,C 180,E1 -20084.272,E2 -20084.272} C_VEL
LIN {X 0,Y 228.005,Z 251.088,A -85,B 0,C 180,E1 -20087.953,E2 -20087.953} C_VEL
LIN {X 0,Y 227.925,Z 251.084,A -85,B 0,C 180,E1 -20092.324,E2 -20092.324} C_VEL
LIN {X 0,Y 227.924,Z 251.091,A -85,B 0,C 180,E1 -20096.592,E2 -20096.592} C_VEL
LIN {X 0,Y 227.875,Z 251.099,A -85,B 0,C 180,E1 -20100.28,E2 -20100.28} C_VEL
LIN {X 0,Y 227.877,Z 251.096,A -85,B 0,C 180,E1 -20103.72,E2 -20103.72} C_VEL
LIN {X 0,Y 227.844,Z 251.103,A -85,B 0,C 180,E1 -20108.09,E2 -20108.09} C_VEL
LIN {X 0,Y 227.806,Z 251.098,A -85,B 0,C 180,E1 -20112.743,E2 -20112.743} C_VEL
LIN {X 0,Y 227.809,Z 251.104,A -85,B 0,C 180,E1 -20117.257,E2 -20117.257} C_VEL
LIN {X 0,Y 227.843,Z 251.095,A -85,B 0,C 180,E1 -20121.908,E2 -20121.908} C_VEL
LIN {X 0,Y 227.879,Z 251.088,A -85,B 0,C 180,E1 -20126.377,E2 -20126.377} C_VEL
LIN {X 0,Y 227.903,Z 251.095,A -85,B 0,C 180,E1 -20130.435,E2 -20130.435} C_VEL
LIN {X 0,Y 227.927,Z 251.075,A -85,B 0,C 180,E1 -20134.425,E2 -20134.425} C_VEL
LIN {X 0,Y 227.961,Z 251.074,A -85,B 0,C 180,E1 -20138.287,E2 -20138.287} C_VEL
LIN {X 0,Y 228.034,Z 251.078,A -85,B 0,C 180,E1 -20142.825,E2 -20142.825} C_VEL
LIN {X 0,Y 228.092,Z 251.053,A -85,B 0,C 180,E1 -20147.544,E2 -20147.544} C_VEL
LIN {X 0,Y 228.324,Z 251.029,A -85,B 0,C 180,E1 -20151.147,E2 -20151.147} C_VEL
LIN {X 0,Y 228.357,Z 251.034,A -85,B 0,C 180,E1 -20152.928,E2 -20152.928} C_VEL
LIN {X 0,Y 228.553,Z 251.009,A -85,B 0,C 180,E1 -20158.238,E2 -20158.238} C_VEL
LIN {X 0,Y 228.553,Z 250.992,A -85,B 0,C 180,E1 -20161.762,E2 -20161.762} C_VEL
LIN {X 0,Y 228.357,Z 251.038,A -85,B 0,C 180,E1 -20167.071,E2 -20167.071} C_VEL
LIN {X 0,Y 228.166,Z 251.056,A -85,B 0,C 180,E1 -20170.65,E2 -20170.65} C_VEL
LIN {X 0,Y 228.063,Z 251.058,A -85,B 0,C 180,E1 -20174.272,E2 -20174.272} C_VEL
LIN {X 0,Y 228.002,Z 251.083,A -85,B 0,C 180,E1 -20177.953,E2 -20177.953} C_VEL
LIN {X 0,Y 227.929,Z 251.085,A -85,B 0,C 180,E1 -20182.329,E2 -20182.329} C_VEL
LIN {X 0,Y 227.904,Z 251.093,A -85,B 0,C 180,E1 -20187.101,E2 -20187.101} C_VEL
LIN {X 0,Y 227.907,Z 251.094,A -85,B 0,C 180,E1 -20190.296,E2 -20190.296} C_VEL
LIN {X 0,Y 227.837,Z 251.097,A -85,B 0,C 180,E1 -20194.77,E2 -20194.77} C_VEL
LIN {X 0,Y 227.17,Z 251.19,A -85,B 0,C 180,E1 -20196.246,E2 -20196.246} C_VEL
LIN {X 0,Y 224.3,Z 251.544,A -85,B 0,C 180,E1 -20198.655,E2 -20198.655} C_VEL
LIN {X 0,Y 221.865,Z 251.846,A -85,B 0,C 180,E1 -20200.621,E2 -20200.621} C_VEL
LIN {X 0,Y 220.833,Z 251.966,A -85,B 0,C 180,E1 -20202.148,E2 -20202.148} C_VEL
LIN {X 0,Y 220.756,Z 251.974,A -85,B 0,C 180,E1 -20202.665,E2 -20202.665} C_VEL
LIN {X 0,Y 220.768,Z 251.986,A -85,B 0,C 180,E1 -20207.07,E2 -20207.07} C_VEL
LIN {X 0,Y 220.868,Z 252.128,A -85,B 0,C 180,E1 -20210.689,E2 -20210.689} C_VEL
LIN {X 0,Y 223.07,Z 261.378,A -85,B 0,C 180,E1 -20215,E2 -20215} C_VEL
LIN {X 0,Y 223.223,Z 262.031,A -85,B 0,C 180,E1 -20215.197,E2 -20215.197} C_VEL
LIN {X 0,Y 232.267,Z 283.749,A -85,B 0,C 180,E1 -20217.276,E2 -20217.276} C_VEL
LIN {X 0,Y 234.987,Z 291.128,A -85,B 0,C 180,E1 -20217.895,E2 -20217.895} C_VEL
LIN {X 0,Y 238.156,Z 314.368,A -85,B 0,C 180,E1 -20219.108,E2 -20219.108} C_VEL
LIN {X 0,Y 235.813,Z 371.23,A -85,B 0,C 180,E1 -20220.883,E2 -20220.883} C_VEL
LIN {X 0,Y 234.491,Z 385.055,A -85,B 0,C 180,E1 -20221.65,E2 -20221.65} C_VEL
LIN {X 0,Y 233.082,Z 396.731,A -85,B 0,C 180,E1 -20222.625,E2 -20222.625} C_VEL
LIN {X 0,Y 231.29,Z 407.843,A -85,B 0,C 180,E1 -20223.858,E2 -20223.858} C_VEL
LIN {X 0,Y 229.037,Z 419.438,A -85,B 0,C 180,E1 -20225.529,E2 -20225.529} C_VEL
LIN {X 0,Y 226.829,Z 429.903,A -85,B 0,C 180,E1 -20227.455,E2 -20227.455} C_VEL
LIN {X 0,Y 224.839,Z 439.4,A -85,B 0,C 180,E1 -20229.675,E2 -20229.675} C_VEL
LIN {X 0,Y 222.96,Z 447.726,A -85,B 0,C 180,E1 -20232.102,E2 -20232.102} C_VEL
LIN {X 0,Y 221.26,Z 455.159,A -85,B 0,C 180,E1 -20234.809,E2 -20234.809} C_VEL
LIN {X 0,Y 220.093,Z 460.187,A -85,B 0,C 180,E1 -20237.084,E2 -20237.084} C_VEL
LIN {X 0,Y 219.274,Z 465.065,A -85,B 0,C 180,E1 -20239.847,E2 -20239.847} C_VEL
LIN {X 0,Y 218.758,Z 468.79,A -85,B 0,C 180,E1 -20242.617,E2 -20242.617} C_VEL
LIN {X 0,Y 218.52,Z 471.619,A -85,B 0,C 180,E1 -20245.575,E2 -20245.575} C_VEL
LIN {X 0,Y 218.562,Z 473.186,A -85,B 0,C 180,E1 -20248.158,E2 -20248.158} C_VEL
LIN {X 0,Y 218.648,Z 473.809,A -85,B 0,C 180,E1 -20250,E2 -20250} C_VEL
LIN {X 0,Y 218.552,Z 474.033,A -85,B 0,C 180,E1 -20251.843,E2 -20251.843} C_VEL
LIN {X 0,Y 218.513,Z 473.637,A -85,B 0,C 180,E1 -20254.403,E2 -20254.403} C_VEL
LIN {X 0,Y 218.76,Z 472.232,A -85,B 0,C 180,E1 -20257.384,E2 -20257.384} C_VEL
LIN {X 0,Y 219.096,Z 470.845,A -85,B 0,C 180,E1 -20259.23,E2 -20259.23} C_VEL
LIN {X 0,Y 219.968,Z 467.938,A -85,B 0,C 180,E1 -20261.986,E2 -20261.986} C_VEL
LIN {X 0,Y 221.178,Z 464.018,A -85,B 0,C 180,E1 -20264.726,E2 -20264.726} C_VEL
LIN {X 0,Y 223.09,Z 458.984,A -85,B 0,C 180,E1 -20267.414,E2 -20267.414} C_VEL
LIN {X 0,Y 225.305,Z 452.688,A -85,B 0,C 180,E1 -20270.068,E2 -20270.068} C_VEL
LIN {X 0,Y 227.959,Z 444.84,A -85,B 0,C 180,E1 -20272.667,E2 -20272.667} C_VEL
LIN {X 0,Y 230.541,Z 436.881,A -85,B 0,C 180,E1 -20274.782,E2 -20274.782} C_VEL
LIN {X 0,Y 233.567,Z 427.204,A -85,B 0,C 180,E1 -20276.83,E2 -20276.83} C_VEL
LIN {X 0,Y 236.582,Z 416.489,A -85,B 0,C 180,E1 -20278.621,E2 -20278.621} C_VEL
LIN {X 0,Y 239.066,Z 406.116,A -85,B 0,C 180,E1 -20279.984,E2 -20279.984} C_VEL
LIN {X 0,Y 241.467,Z 393.738,A -85,B 0,C 180,E1 -20281.228,E2 -20281.228} C_VEL
LIN {X 0,Y 243.46,Z 380.811,A -85,B 0,C 180,E1 -20282.157,E2 -20282.157} C_VEL
LIN {X 0,Y 244.779,Z 368.2,A -85,B 0,C 180,E1 -20282.754,E2 -20282.754} C_VEL
LIN {X 0,Y 247.315,Z 316.583,A -85,B 0,C 180,E1 -20284.323,E2 -20284.323} C_VEL
LIN {X 0,Y 245.425,Z 302.542,A -85,B 0,C 180,E1 -20285.24,E2 -20285.24} C_VEL
LIN {X 0,Y 238.879,Z 287.586,A -85,B 0,C 180,E1 -20287.231,E2 -20287.231} C_VEL
LIN {X 0,Y 232.106,Z 274.566,A -85,B 0,C 180,E1 -20289.391,E2 -20289.391} C_VEL
LIN {X 0,Y 228.771,Z 269.053,A -85,B 0,C 180,E1 -20290.506,E2 -20290.506} C_VEL
LIN {X 0,Y 226.23,Z 264.786,A -85,B 0,C 180,E1 -20291.406,E2 -20291.406} C_VEL
LIN {X 0,Y 223.514,Z 260.518,A -85,B 0,C 180,E1 -20292.392,E2 -20292.392} C_VEL
LIN {X 0,Y 223.135,Z 259.616,A -85,B 0,C 180,E1 -20292.642,E2 -20292.642} C_VEL
LIN {X 0,Y 221.607,Z 254.619,A -85,B 0,C 180,E1 -20295.757,E2 -20295.757} C_VEL
LIN {X 0,Y 220.782,Z 251.979,A -85,B 0,C 180,E1 -20297.656,E2 -20297.656} C_VEL
LIN {X 0,Y 220.807,Z 251.977,A -85,B 0,C 180,E1 -20300.463,E2 -20300.463} C_VEL
LIN {X 0,Y 220.802,Z 251.971,A -85,B 0,C 180,E1 -20305.045,E2 -20305.045} C_VEL
LIN {X 0,Y 220.869,Z 251.963,A -85,B 0,C 180,E1 -20309.395,E2 -20309.395} C_VEL
LIN {X 0,Y 220.896,Z 251.96,A -85,B 0,C 180,E1 -20313.55,E2 -20313.55} C_VEL
LIN {X 0,Y 220.879,Z 251.961,A -85,B 0,C 180,E1 -20317.554,E2 -20317.554} C_VEL
LIN {X 0,Y 220.985,Z 251.95,A -85,B 0,C 180,E1 -20322.571,E2 -20322.571} C_VEL
LIN {X 0,Y 221.026,Z 251.943,A -85,B 0,C 180,E1 -20327.139,E2 -20327.139} C_VEL
LIN {X 0,Y 221.236,Z 251.913,A -85,B 0,C 180,E1 -20330.861,E2 -20330.861} C_VEL
LIN {X 0,Y 221.289,Z 251.92,A -85,B 0,C 180,E1 -20332.702,E2 -20332.702} C_VEL
LIN {X 0,Y 221.513,Z 251.889,A -85,B 0,C 180,E1 -20338.182,E2 -20338.182} C_VEL
LIN {X 0,Y 221.513,Z 251.893,A -85,B 0,C 180,E1 -20341.818,E2 -20341.818} C_VEL
LIN {X 0,Y 221.29,Z 251.912,A -85,B 0,C 180,E1 -20347.299,E2 -20347.299} C_VEL
LIN {X 0,Y 221.108,Z 251.937,A -85,B 0,C 180,E1 -20350.995,E2 -20350.995} C_VEL
LIN {X 0,Y 221.017,Z 251.954,A -85,B 0,C 180,E1 -20356.63,E2 -20356.63} C_VEL
LIN {X 0,Y 220.935,Z 252.162,A -85,B 0,C 180,E1 -20361.826,E2 -20361.826} C_VEL
LIN {X 0,Y 222.132,Z 255.187,A -85,B 0,C 180,E1 -20362.377,E2 -20362.377} C_VEL
LIN {X 0,Y 224.295,Z 257.493,A -85,B 0,C 180,E1 -20363.131,E2 -20363.131} C_VEL
LIN {X 0,Y 226.464,Z 260.86,A -85,B 0,C 180,E1 -20363.915,E2 -20363.915} C_VEL
LIN {X 0,Y 227.95,Z 262.714,A -85,B 0,C 180,E1 -20364.415,E2 -20364.415} C_VEL
LIN {X 0,Y 233.306,Z 271.232,A -85,B 0,C 180,E1 -20366.2,E2 -20366.2} C_VEL
LIN {X 0,Y 239.809,Z 282.979,A -85,B 0,C 180,E1 -20368.224,E2 -20368.224} C_VEL
LIN {X 0,Y 245.538,Z 295.107,A -85,B 0,C 180,E1 -20369.93,E2 -20369.93} C_VEL
LIN {X 0,Y 248.064,Z 301.168,A -85,B 0,C 180,E1 -20370.662,E2 -20370.662} C_VEL
LIN {X 0,Y 245.025,Z 358.905,A -85,B 0,C 180,E1 -20372.395,E2 -20372.395} C_VEL
LIN {X 0,Y 243.692,Z 371.908,A -85,B 0,C 180,E1 -20373.067,E2 -20373.067} C_VEL
LIN {X 0,Y 241.806,Z 384.886,A -85,B 0,C 180,E1 -20374.072,E2 -20374.072} C_VEL
LIN {X 0,Y 239.623,Z 396.609,A -85,B 0,C 180,E1 -20375.332,E2 -20375.332} C_VEL
LIN {X 0,Y 237.08,Z 407.446,A -85,B 0,C 180,E1 -20376.833,E2 -20376.833} C_VEL
LIN {X 0,Y 234.201,Z 418.119,A -85,B 0,C 180,E1 -20378.72,E2 -20378.72} C_VEL
LIN {X 0,Y 231.537,Z 426.786,A -85,B 0,C 180,E1 -20380.638,E2 -20380.638} C_VEL
LIN {X 0,Y 228.567,Z 435.59,A -85,B 0,C 180,E1 -20383.091,E2 -20383.091} C_VEL
LIN {X 0,Y 225.959,Z 442.897,A -85,B 0,C 180,E1 -20385.674,E2 -20385.674} C_VEL
LIN {X 0,Y 223.478,Z 449.5,A -85,B 0,C 180,E1 -20388.669,E2 -20388.669} C_VEL
LIN {X 0,Y 221.502,Z 454.567,A -85,B 0,C 180,E1 -20391.759,E2 -20391.759} C_VEL
LIN {X 0,Y 220.077,Z 458.262,A -85,B 0,C 180,E1 -20394.913,E2 -20394.913} C_VEL
LIN {X 0,Y 219.403,Z 460.013,A -85,B 0,C 180,E1 -20397.006,E2 -20397.006} C_VEL
LIN {X 0,Y 218.565,Z 461.635,A -85,B 0,C 180,E1 -20400.25,E2 -20400.25} C_VEL
LIN {X 0,Y 218.229,Z 462.04,A -85,B 0,C 180,E1 -20403.201,E2 -20403.201} C_VEL
LIN {X 0,Y 218.154,Z 461.708,A -85,B 0,C 180,E1 -20405.241,E2 -20405.241} C_VEL
LIN {X 0,Y 218.206,Z 460.935,A -85,B 0,C 180,E1 -20407.263,E2 -20407.263} C_VEL
LIN {X 0,Y 218.448,Z 459.658,A -85,B 0,C 180,E1 -20409.274,E2 -20409.274} C_VEL
LIN {X 0,Y 219.064,Z 456.84,A -85,B 0,C 180,E1 -20412.255,E2 -20412.255} C_VEL
LIN {X 0,Y 219.803,Z 452.916,A -85,B 0,C 180,E1 -20415.179,E2 -20415.179} C_VEL
LIN {X 0,Y 220.9,Z 447.763,A -85,B 0,C 180,E1 -20418.065,E2 -20418.065} C_VEL
LIN {X 0,Y 222.453,Z 441.218,A -85,B 0,C 180,E1 -20420.911,E2 -20420.911} C_VEL
LIN {X 0,Y 224.03,Z 434.496,A -85,B 0,C 180,E1 -20423.244,E2 -20423.244} C_VEL
LIN {X 0,Y 226.178,Z 425.295,A -85,B 0,C 180,E1 -20425.798,E2 -20425.798} C_VEL
LIN {X 0,Y 228.342,Z 415.231,A -85,B 0,C 180,E1 -20428.015,E2 -20428.015} C_VEL
LIN {X 0,Y 230.375,Z 405.159,A -85,B 0,C 180,E1 -20429.781,E2 -20429.781} C_VEL
LIN {X 0,Y 232.363,Z 393.394,A -85,B 0,C 180,E1 -20431.399,E2 -20431.399} C_VEL
LIN {X 0,Y 234.031,Z 381.075,A -85,B 0,C 180,E1 -20432.689,E2 -20432.689} C_VEL
LIN {X 0,Y 235.357,Z 368.093,A -85,B 0,C 180,E1 -20433.669,E2 -20433.669} C_VEL
LIN {X 0,Y 236.249,Z 355.131,A -85,B 0,C 180,E1 -20434.29,E2 -20434.29} C_VEL
LIN {X 0,Y 238.835,Z 293.824,A -85,B 0,C 180,E1 -20436.145,E2 -20436.145} C_VEL
LIN {X 0,Y 234.067,Z 280.467,A -85,B 0,C 180,E1 -20437.221,E2 -20437.221} C_VEL
LIN {X 0,Y 224.873,Z 259.427,A -85,B 0,C 180,E1 -20439.278,E2 -20439.278} C_VEL
LIN {X 0,Y 221.382,Z 252.951,A -85,B 0,C 180,E1 -20440.043,E2 -20440.043} C_VEL
LIN {X 0,Y 221.15,Z 251.934,A -85,B 0,C 180,E1 -20440.142,E2 -20440.142} C_VEL
LIN {X 0,Y 220.999,Z 251.961,A -85,B 0,C 180,E1 -20444.738,E2 -20444.738} C_VEL
LIN {X 0,Y 220.923,Z 251.969,A -85,B 0,C 180,E1 -20448.549,E2 -20448.549} C_VEL
LIN {X 0,Y 220.872,Z 251.961,A -85,B 0,C 180,E1 -20452.666,E2 -20452.666} C_VEL
LIN {X 0,Y 220.867,Z 251.97,A -85,B 0,C 180,E1 -20457.005,E2 -20457.005} C_VEL
LIN {X 0,Y 220.819,Z 251.978,A -85,B 0,C 180,E1 -20460.758,E2 -20460.758} C_VEL
LIN {X 0,Y 220.802,Z 251.97,A -85,B 0,C 180,E1 -20464.954,E2 -20464.954} C_VEL
LIN {X 0,Y 220.806,Z 251.981,A -85,B 0,C 180,E1 -20469.536,E2 -20469.536} C_VEL
LIN {X 0,Y 220.77,Z 251.969,A -85,B 0,C 180,E1 -20474.454,E2 -20474.454} C_VEL
LIN {X 0,Y 220.769,Z 251.986,A -85,B 0,C 180,E1 -20478.047,E2 -20478.047} C_VEL
LIN {X 0,Y 220.824,Z 251.964,A -85,B 0,C 180,E1 -20482.792,E2 -20482.792} C_VEL
LIN {X 0,Y 220.816,Z 251.971,A -85,B 0,C 180,E1 -20487.243,E2 -20487.243} C_VEL
LIN {X 0,Y 220.826,Z 251.975,A -85,B 0,C 180,E1 -20491.485,E2 -20491.485} C_VEL
LIN {X 0,Y 220.866,Z 251.948,A -85,B 0,C 180,E1 -20495.565,E2 -20495.565} C_VEL
LIN {X 0,Y 220.892,Z 251.96,A -85,B 0,C 180,E1 -20499.514,E2 -20499.514} C_VEL
LIN {X 0,Y 221.015,Z 251.952,A -85,B 0,C 180,E1 -20503.37,E2 -20503.37} C_VEL
LIN {X 0,Y 221.116,Z 251.911,A -85,B 0,C 180,E1 -20509.006,E2 -20509.006} C_VEL
LIN {X 0,Y 221.31,Z 251.913,A -85,B 0,C 180,E1 -20512.702,E2 -20512.702} C_VEL
LIN {X 0,Y 221.511,Z 251.886,A -85,B 0,C 180,E1 -20518.182,E2 -20518.182} C_VEL
LIN {X 0,Y 221.511,Z 251.867,A -85,B 0,C 180,E1 -20521.818,E2 -20521.818} C_VEL
LIN {X 0,Y 221.31,Z 251.915,A -85,B 0,C 180,E1 -20527.298,E2 -20527.298} C_VEL
LIN {X 0,Y 221.11,Z 251.933,A -85,B 0,C 180,E1 -20530.994,E2 -20530.994} C_VEL
LIN {X 0,Y 221.015,Z 251.951,A -85,B 0,C 180,E1 -20536.63,E2 -20536.63} C_VEL
LIN {X 0,Y 220.891,Z 251.965,A -85,B 0,C 180,E1 -20540.486,E2 -20540.486} C_VEL
LIN {X 0,Y 220.866,Z 251.972,A -85,B 0,C 180,E1 -20544.435,E2 -20544.435} C_VEL
LIN {X 0,Y 220.835,Z 251.97,A -85,B 0,C 180,E1 -20548.514,E2 -20548.514} C_VEL
LIN {X 0,Y 220.816,Z 251.975,A -85,B 0,C 180,E1 -20552.756,E2 -20552.756} C_VEL
LIN {X 0,Y 220.809,Z 251.977,A -85,B 0,C 180,E1 -20557.279,E2 -20557.279} C_VEL
LIN {X 0,Y 220.793,Z 251.983,A -85,B 0,C 180,E1 -20560.188,E2 -20560.188} C_VEL
LIN {X 0,Y 220.756,Z 251.974,A -85,B 0,C 180,E1 -20562.665,E2 -20562.665} C_VEL
LIN {X 0,Y 220.079,Z 252.063,A -85,B 0,C 180,E1 -20563.676,E2 -20563.676} C_VEL
LIN {X 0,Y 217.213,Z 252.43,A -85,B 0,C 180,E1 -20565.262,E2 -20565.262} C_VEL
LIN {X 0,Y 214.327,Z 252.788,A -85,B 0,C 180,E1 -20566.889,E2 -20566.889} C_VEL
LIN {X 0,Y 213.664,Z 252.864,A -85,B 0,C 180,E1 -20567.946,E2 -20567.946} C_VEL
LIN {X 0,Y 213.796,Z 252.979,A -85,B 0,C 180,E1 -20569.892,E2 -20569.892} C_VEL
LIN {X 0,Y 215.86,Z 261.491,A -85,B 0,C 180,E1 -20574.024,E2 -20574.024} C_VEL
LIN {X 0,Y 224.445,Z 281.751,A -85,B 0,C 180,E1 -20576.13,E2 -20576.13} C_VEL
LIN {X 0,Y 228.746,Z 293.053,A -85,B 0,C 180,E1 -20577.152,E2 -20577.152} C_VEL
LIN {X 0,Y 231.756,Z 315.765,A -85,B 0,C 180,E1 -20578.377,E2 -20578.377} C_VEL
LIN {X 0,Y 229.444,Z 370.271,A -85,B 0,C 180,E1 -20580.111,E2 -20580.111} C_VEL
LIN {X 0,Y 228.172,Z 383.698,A -85,B 0,C 180,E1 -20580.854,E2 -20580.854} C_VEL
LIN {X 0,Y 226.618,Z 396.238,A -85,B 0,C 180,E1 -20581.901,E2 -20581.901} C_VEL
LIN {X 0,Y 224.857,Z 406.597,A -85,B 0,C 180,E1 -20583.051,E2 -20583.051} C_VEL
LIN {X 0,Y 222.583,Z 418.418,A -85,B 0,C 180,E1 -20584.77,E2 -20584.77} C_VEL
LIN {X 0,Y 220.299,Z 429.027,A -85,B 0,C 180,E1 -20586.748,E2 -20586.748} C_VEL
LIN {X 0,Y 218.344,Z 437.704,A -85,B 0,C 180,E1 -20588.771,E2 -20588.771} C_VEL
LIN {X 0,Y 216.595,Z 445.707,A -85,B 0,C 180,E1 -20591.067,E2 -20591.067} C_VEL
LIN {X 0,Y 214.645,Z 453.481,A -85,B 0,C 180,E1 -20593.841,E2 -20593.841} C_VEL
LIN {X 0,Y 213.134,Z 459.706,A -85,B 0,C 180,E1 -20596.655,E2 -20596.655} C_VEL
LIN {X 0,Y 212.242,Z 464.646,A -85,B 0,C 180,E1 -20599.507,E2 -20599.507} C_VEL
LIN {X 0,Y 211.687,Z 468.428,A -85,B 0,C 180,E1 -20602.369,E2 -20602.369} C_VEL
LIN {X 0,Y 211.419,Z 471.564,A -85,B 0,C 180,E1 -20605.759,E2 -20605.759} C_VEL
LIN {X 0,Y 211.461,Z 472.926,A -85,B 0,C 180,E1 -20608.096,E2 -20608.096} C_VEL
LIN {X 0,Y 211.563,Z 473.574,A -85,B 0,C 180,E1 -20610,E2 -20610} C_VEL
LIN {X 0,Y 211.451,Z 473.822,A -85,B 0,C 180,E1 -20611.905,E2 -20611.905} C_VEL
LIN {X 0,Y 211.419,Z 473.56,A -85,B 0,C 180,E1 -20614.242,E2 -20614.242} C_VEL
LIN {X 0,Y 211.689,Z 472.119,A -85,B 0,C 180,E1 -20617.632,E2 -20617.632} C_VEL
LIN {X 0,Y 212.07,Z 470.757,A -85,B 0,C 180,E1 -20619.538,E2 -20619.538} C_VEL
LIN {X 0,Y 212.989,Z 467.902,A -85,B 0,C 180,E1 -20622.385,E2 -20622.385} C_VEL
LIN {X 0,Y 214.302,Z 464.035,A -85,B 0,C 180,E1 -20625.21,E2 -20625.21} C_VEL
LIN {X 0,Y 216.321,Z 459.066,A -85,B 0,C 180,E1 -20627.978,E2 -20627.978} C_VEL
LIN {X 0,Y 218.652,Z 452.85,A -85,B 0,C 180,E1 -20630.706,E2 -20630.706} C_VEL
LIN {X 0,Y 221.423,Z 445.141,A -85,B 0,C 180,E1 -20633.375,E2 -20633.375} C_VEL
LIN {X 0,Y 224.134,Z 437.285,A -85,B 0,C 180,E1 -20635.541,E2 -20635.541} C_VEL
LIN {X 0,Y 227.667,Z 426.657,A -85,B 0,C 180,E1 -20637.834,E2 -20637.834} C_VEL
LIN {X 0,Y 230.397,Z 417.159,A -85,B 0,C 180,E1 -20639.464,E2 -20639.464} C_VEL
LIN {X 0,Y 232.989,Z 407,A -85,B 0,C 180,E1 -20640.85,E2 -20640.85} C_VEL
LIN {X 0,Y 235.511,Z 395.034,A -85,B 0,C 180,E1 -20642.11,E2 -20642.11} C_VEL
LIN {X 0,Y 237.635,Z 381.883,A -85,B 0,C 180,E1 -20643.107,E2 -20643.107} C_VEL
LIN {X 0,Y 239.116,Z 368.925,A -85,B 0,C 180,E1 -20643.758,E2 -20643.758} C_VEL
LIN {X 0,Y 241.806,Z 317.673,A -85,B 0,C 180,E1 -20645.351,E2 -20645.351} C_VEL
LIN {X 0,Y 240.278,Z 305.645,A -85,B 0,C 180,E1 -20646.164,E2 -20646.164} C_VEL
LIN {X 0,Y 234.067,Z 291.248,A -85,B 0,C 180,E1 -20648.159,E2 -20648.159} C_VEL
LIN {X 0,Y 227.903,Z 279.176,A -85,B 0,C 180,E1 -20650.25,E2 -20650.25} C_VEL
LIN {X 0,Y 222.452,Z 269.982,A -85,B 0,C 180,E1 -20652.212,E2 -20652.212} C_VEL
LIN {X 0,Y 218.894,Z 264.433,A -85,B 0,C 180,E1 -20653.577,E2 -20653.577} C_VEL
LIN {X 0,Y 215.876,Z 259.754,A -85,B 0,C 180,E1 -20654.819,E2 -20654.819} C_VEL
LIN {X 0,Y 214.955,Z 256.856,A -85,B 0,C 180,E1 -20656.638,E2 -20656.638} C_VEL
LIN {X 0,Y 213.746,Z 252.863,A -85,B 0,C 180,E1 -20659.661,E2 -20659.661} C_VEL
LIN {X 0,Y 213.744,Z 252.856,A -85,B 0,C 180,E1 -20663.712,E2 -20663.712} C_VEL
LIN {X 0,Y 213.768,Z 252.846,A -85,B 0,C 180,E1 -20668.263,E2 -20668.263} C_VEL
LIN {X 0,Y 213.827,Z 252.837,A -85,B 0,C 180,E1 -20672.603,E2 -20672.603} C_VEL
LIN {X 0,Y 213.853,Z 252.834,A -85,B 0,C 180,E1 -20676.953,E2 -20676.953} C_VEL
LIN {X 0,Y 213.944,Z 252.829,A -85,B 0,C 180,E1 -20682.804,E2 -20682.804} C_VEL
LIN {X 0,Y 213.981,Z 252.817,A -85,B 0,C 180,E1 -20686.708,E2 -20686.708} C_VEL
LIN {X 0,Y 214.168,Z 252.793,A -85,B 0,C 180,E1 -20690.556,E2 -20690.556} C_VEL
LIN {X 0,Y 214.227,Z 252.798,A -85,B 0,C 180,E1 -20692.46,E2 -20692.46} C_VEL
LIN {X 0,Y 214.446,Z 252.77,A -85,B 0,C 180,E1 -20698.122,E2 -20698.122} C_VEL
LIN {X 0,Y 214.547,Z 252.747,A -85,B 0,C 180,E1 -20700,E2 -20700} C_VEL
LIN {X 0,Y 214.446,Z 252.773,A -85,B 0,C 180,E1 -20701.878,E2 -20701.878} C_VEL
LIN {X 0,Y 214.228,Z 252.79,A -85,B 0,C 180,E1 -20707.541,E2 -20707.541} C_VEL
LIN {X 0,Y 214.024,Z 252.817,A -85,B 0,C 180,E1 -20711.363,E2 -20711.363} C_VEL
LIN {X 0,Y 213.934,Z 252.829,A -85,B 0,C 180,E1 -20715.237,E2 -20715.237} C_VEL
LIN {X 0,Y 213.848,Z 252.846,A -85,B 0,C 180,E1 -20719.499,E2 -20719.499} C_VEL
LIN {X 0,Y 214.707,Z 255.432,A -85,B 0,C 180,E1 -20719.978,E2 -20719.978} C_VEL
LIN {X 0,Y 216.669,Z 257.679,A -85,B 0,C 180,E1 -20720.78,E2 -20720.78} C_VEL
LIN {X 0,Y 217.565,Z 258.527,A -85,B 0,C 180,E1 -20721.124,E2 -20721.124} C_VEL
LIN {X 0,Y 219.527,Z 261.663,A -85,B 0,C 180,E1 -20721.919,E2 -20721.919} C_VEL
LIN {X 0,Y 221.058,Z 263.574,A -85,B 0,C 180,E1 -20722.491,E2 -20722.491} C_VEL
LIN {X 0,Y 223.659,Z 267.143,A -85,B 0,C 180,E1 -20723.443,E2 -20723.443} C_VEL
LIN {X 0,Y 229.149,Z 275.934,A -85,B 0,C 180,E1 -20725.368,E2 -20725.368} C_VEL
LIN {X 0,Y 235.207,Z 287.064,A -85,B 0,C 180,E1 -20727.368,E2 -20727.368} C_VEL
LIN {X 0,Y 240.696,Z 298.872,A -85,B 0,C 180,E1 -20729.086,E2 -20729.086} C_VEL
LIN {X 0,Y 242.481,Z 303.188,A -85,B 0,C 180,E1 -20729.638,E2 -20729.638} C_VEL
LIN {X 0,Y 239.329,Z 360.003,A -85,B 0,C 180,E1 -20731.396,E2 -20731.396} C_VEL
LIN {X 0,Y 237.843,Z 373.821,A -85,B 0,C 180,E1 -20732.161,E2 -20732.161} C_VEL
LIN {X 0,Y 235.912,Z 386.031,A -85,B 0,C 180,E1 -20733.153,E2 -20733.153} C_VEL
LIN {X 0,Y 233.479,Z 398.135,A -85,B 0,C 180,E1 -20734.512,E2 -20734.512} C_VEL
LIN {X 0,Y 230.692,Z 409.45,A -85,B 0,C 180,E1 -20736.165,E2 -20736.165} C_VEL
LIN {X 0,Y 227.617,Z 419.972,A -85,B 0,C 180,E1 -20738.136,E2 -20738.136} C_VEL
LIN {X 0,Y 224.283,Z 430,A -85,B 0,C 180,E1 -20740.546,E2 -20740.546} C_VEL
LIN {X 0,Y 221.288,Z 438.259,A -85,B 0,C 180,E1 -20743.074,E2 -20743.074} C_VEL
LIN {X 0,Y 218.256,Z 446.049,A -85,B 0,C 180,E1 -20746.186,E2 -20746.186} C_VEL
LIN {X 0,Y 215.811,Z 452.077,A -85,B 0,C 180,E1 -20749.359,E2 -20749.359} C_VEL
LIN {X 0,Y 213.879,Z 456.766,A -85,B 0,C 180,E1 -20752.789,E2 -20752.789} C_VEL
LIN {X 0,Y 212.642,Z 459.635,A -85,B 0,C 180,E1 -20755.815,E2 -20755.815} C_VEL
LIN {X 0,Y 211.987,Z 461.025,A -85,B 0,C 180,E1 -20757.964,E2 -20757.964} C_VEL
LIN {X 0,Y 211.499,Z 461.874,A -85,B 0,C 180,E1 -20760.103,E2 -20760.103} C_VEL
LIN {X 0,Y 211.202,Z 462.217,A -85,B 0,C 180,E1 -20762.234,E2 -20762.234} C_VEL
LIN {X 0,Y 211.094,Z 462.099,A -85,B 0,C 180,E1 -20764.354,E2 -20764.354} C_VEL
LIN {X 0,Y 211.07,Z 461.455,A -85,B 0,C 180,E1 -20766.449,E2 -20766.449} C_VEL
LIN {X 0,Y 211.248,Z 460.274,A -85,B 0,C 180,E1 -20768.676,E2 -20768.676} C_VEL
LIN {X 0,Y 211.776,Z 457.813,A -85,B 0,C 180,E1 -20771.623,E2 -20771.623} C_VEL
LIN {X 0,Y 212.541,Z 454.164,A -85,B 0,C 180,E1 -20774.661,E2 -20774.661} C_VEL
LIN {X 0,Y 213.605,Z 449.313,A -85,B 0,C 180,E1 -20777.651,E2 -20777.651} C_VEL
LIN {X 0,Y 215.07,Z 443.087,A -85,B 0,C 180,E1 -20780.596,E2 -20780.596} C_VEL
LIN {X 0,Y 217.006,Z 435.278,A -85,B 0,C 180,E1 -20783.491,E2 -20783.491} C_VEL
LIN {X 0,Y 219.007,Z 427.177,A -85,B 0,C 180,E1 -20785.882,E2 -20785.882} C_VEL
LIN {X 0,Y 221.169,Z 417.469,A -85,B 0,C 180,E1 -20788.179,E2 -20788.179} C_VEL
LIN {X 0,Y 223.476,Z 406.534,A -85,B 0,C 180,E1 -20790.215,E2 -20790.215} C_VEL
LIN {X 0,Y 225.369,Z 395.887,A -85,B 0,C 180,E1 -20791.787,E2 -20791.787} C_VEL
LIN {X 0,Y 227.134,Z 384.333,A -85,B 0,C 180,E1 -20793.104,E2 -20793.104} C_VEL
LIN {X 0,Y 228.564,Z 371.419,A -85,B 0,C 180,E1 -20794.188,E2 -20794.188} C_VEL
LIN {X 0,Y 229.675,Z 357.916,A -85,B 0,C 180,E1 -20794.937,E2 -20794.937} C_VEL
LIN {X 0,Y 232.398,Z 294.914,A -85,B 0,C 180,E1 -20796.913,E2 -20796.913} C_VEL
LIN {X 0,Y 227.285,Z 281.277,A -85,B 0,C 180,E1 -20798.103,E2 -20798.103} C_VEL
LIN {X 0,Y 219.353,Z 263.126,A -85,B 0,C 180,E1 -20799.95,E2 -20799.95} C_VEL
LIN {X 0,Y 214.281,Z 253.966,A -85,B 0,C 180,E1 -20801.115,E2 -20801.115} C_VEL
LIN {X 0,Y 214.034,Z 252.825,A -85,B 0,C 180,E1 -20801.264,E2 -20801.264} C_VEL
LIN {X 0,Y 213.936,Z 252.842,A -85,B 0,C 180,E1 -20805.236,E2 -20805.236} C_VEL
LIN {X 0,Y 213.839,Z 252.852,A -85,B 0,C 180,E1 -20809.187,E2 -20809.187} C_VEL
LIN {X 0,Y 213.805,Z 252.842,A -85,B 0,C 180,E1 -20813.231,E2 -20813.231} C_VEL
LIN {X 0,Y 213.789,Z 252.849,A -85,B 0,C 180,E1 -20817.428,E2 -20817.428} C_VEL
LIN {X 0,Y 213.759,Z 252.86,A -85,B 0,C 180,E1 -20821.738,E2 -20821.738} C_VEL
LIN {X 0,Y 213.744,Z 252.849,A -85,B 0,C 180,E1 -20826.288,E2 -20826.288} C_VEL
LIN {X 0,Y 213.711,Z 252.862,A -85,B 0,C 180,E1 -20831.125,E2 -20831.125} C_VEL
LIN {X 0,Y 213.703,Z 252.848,A -85,B 0,C 180,E1 -20833.679,E2 -20833.679} C_VEL
LIN {X 0,Y 213.704,Z 252.859,A -85,B 0,C 180,E1 -20836.344,E2 -20836.344} C_VEL
LIN {X 0,Y 213.717,Z 252.862,A -85,B 0,C 180,E1 -20839.142,E2 -20839.142} C_VEL
LIN {X 0,Y 213.743,Z 252.838,A -85,B 0,C 180,E1 -20843.711,E2 -20843.711} C_VEL
LIN {X 0,Y 213.767,Z 252.855,A -85,B 0,C 180,E1 -20848.262,E2 -20848.262} C_VEL
LIN {X 0,Y 213.825,Z 252.841,A -85,B 0,C 180,E1 -20852.603,E2 -20852.603} C_VEL
LIN {X 0,Y 213.851,Z 252.822,A -85,B 0,C 180,E1 -20856.952,E2 -20856.952} C_VEL
LIN {X 0,Y 213.943,Z 252.833,A -85,B 0,C 180,E1 -20862.803,E2 -20862.803} C_VEL
LIN {X 0,Y 213.979,Z 252.814,A -85,B 0,C 180,E1 -20866.708,E2 -20866.708} C_VEL
LIN {X 0,Y 214.195,Z 252.78,A -85,B 0,C 180,E1 -20870.557,E2 -20870.557} C_VEL
LIN {X 0,Y 214.247,Z 252.789,A -85,B 0,C 180,E1 -20872.46,E2 -20872.46} C_VEL
LIN {X 0,Y 214.445,Z 252.767,A -85,B 0,C 180,E1 -20878.122,E2 -20878.122} C_VEL
LIN {X 0,Y 214.548,Z 252.742,A -85,B 0,C 180,E1 -20880,E2 -20880} C_VEL
LIN {X 0,Y 214.444,Z 252.746,A -85,B 0,C 180,E1 -20881.878,E2 -20881.878} C_VEL
LIN {X 0,Y 214.246,Z 252.796,A -85,B 0,C 180,E1 -20887.54,E2 -20887.54} C_VEL
LIN {X 0,Y 214.04,Z 252.813,A -85,B 0,C 180,E1 -20891.362,E2 -20891.362} C_VEL
LIN {X 0,Y 213.932,Z 252.825,A -85,B 0,C 180,E1 -20895.237,E2 -20895.237} C_VEL
LIN {X 0,Y 213.838,Z 252.847,A -85,B 0,C 180,E1 -20899.187,E2 -20899.187} C_VEL
LIN {X 0,Y 213.846,Z 252.841,A -85,B 0,C 180,E1 -20903.227,E2 -20903.227} C_VEL
LIN {X 0,Y 213.828,Z 252.846,A -85,B 0,C 180,E1 -20907.45,E2 -20907.45} C_VEL
LIN {X 0,Y 213.776,Z 252.856,A -85,B 0,C 180,E1 -20911.736,E2 -20911.736} C_VEL
LIN {X 0,Y 213.742,Z 252.861,A -85,B 0,C 180,E1 -20916.289,E2 -20916.289} C_VEL
LIN {X 0,Y 213.71,Z 252.859,A -85,B 0,C 180,E1 -20921.126,E2 -20921.126} C_VEL
LIN {X 0,Y 213.702,Z 252.856,A -85,B 0,C 180,E1 -20923.68,E2 -20923.68} C_VEL
LIN {X 0,Y 213.664,Z 252.864,A -85,B 0,C 180,E1 -20927.946,E2 -20927.946} C_VEL
LIN {X 0,Y 213.493,Z 253.366,A -85,B 0,C 180,E1 -20928.946,E2 -20928.946} C_VEL
LIN {X 0,Y 213.057,Z 254.676,A -85,B 0,C 180,E1 -20929.893,E2 -20929.893} C_VEL
LIN {X 0,Y 212.246,Z 257.734,A -85,B 0,C 180,E1 -20931.194,E2 -20931.194} C_VEL
LIN {X 0,Y 211.654,Z 261.734,A -85,B 0,C 180,E1 -20932.333,E2 -20932.333} C_VEL
LIN {X 0,Y 211.722,Z 266.381,A -85,B 0,C 180,E1 -20933.292,E2 -20933.292} C_VEL
LIN {X 0,Y 212.694,Z 270.522,A -85,B 0,C 180,E1 -20933.906,E2 -20933.906} C_VEL
LIN {X 0,Y 213.023,Z 271.357,A -85,B 0,C 180,E1 -20934.002,E2 -20934.002} C_VEL
LIN {X 0,Y 220.671,Z 289.8,A -85,B 0,C 180,E1 -20935.9,E2 -20935.9} C_VEL
LIN {X 0,Y 222.739,Z 295.836,A -85,B 0,C 180,E1 -20936.428,E2 -20936.428} C_VEL
LIN {X 0,Y 225.402,Z 315.545,A -85,B 0,C 180,E1 -20937.544,E2 -20937.544} C_VEL
LIN {X 0,Y 223.057,Z 370.009,A -85,B 0,C 180,E1 -20939.327,E2 -20939.327} C_VEL
LIN {X 0,Y 221.715,Z 383.843,A -85,B 0,C 180,E1 -20940.116,E2 -20940.116} C_VEL
LIN {X 0,Y 220.174,Z 395.731,A -85,B 0,C 180,E1 -20941.133,E2 -20941.133} C_VEL
LIN {X 0,Y 218.21,Z 407.006,A -85,B 0,C 180,E1 -20942.421,E2 -20942.421} C_VEL
LIN {X 0,Y 215.859,Z 418.694,A -85,B 0,C 180,E1 -20944.186,E2 -20944.186} C_VEL
LIN {X 0,Y 213.504,Z 429.224,A -85,B 0,C 180,E1 -20946.22,E2 -20946.22} C_VEL
LIN {X 0,Y 211.287,Z 438.704,A -85,B 0,C 180,E1 -20948.538,E2 -20948.538} C_VEL
LIN {X 0,Y 209.464,Z 446.476,A -85,B 0,C 180,E1 -20950.905,E2 -20950.905} C_VEL
LIN {X 0,Y 207.505,Z 454.058,A -85,B 0,C 180,E1 -20953.775,E2 -20953.775} C_VEL
LIN {X 0,Y 205.818,Z 461.049,A -85,B 0,C 180,E1 -20957.177,E2 -20957.177} C_VEL
LIN {X 0,Y 204.993,Z 465.65,A -85,B 0,C 180,E1 -20960.13,E2 -20960.13} C_VEL
LIN {X 0,Y 204.64,Z 468.063,A -85,B 0,C 180,E1 -20962.104,E2 -20962.104} C_VEL
LIN {X 0,Y 204.405,Z 470.032,A -85,B 0,C 180,E1 -20964.08,E2 -20964.08} C_VEL
LIN {X 0,Y 204.336,Z 471.579,A -85,B 0,C 180,E1 -20966.056,E2 -20966.056} C_VEL
LIN {X 0,Y 204.364,Z 472.666,A -85,B 0,C 180,E1 -20968.03,E2 -20968.03} C_VEL
LIN {X 0,Y 204.48,Z 473.34,A -85,B 0,C 180,E1 -20970,E2 -20970} C_VEL
LIN {X 0,Y 204.355,Z 473.611,A -85,B 0,C 180,E1 -20971.971,E2 -20971.971} C_VEL
LIN {X 0,Y 204.347,Z 473.462,A -85,B 0,C 180,E1 -20974.144,E2 -20974.144} C_VEL
LIN {X 0,Y 204.641,Z 472.007,A -85,B 0,C 180,E1 -20977.896,E2 -20977.896} C_VEL
LIN {X 0,Y 205.659,Z 468.939,A -85,B 0,C 180,E1 -20981.832,E2 -20981.832} C_VEL
LIN {X 0,Y 206.913,Z 465.478,A -85,B 0,C 180,E1 -20984.759,E2 -20984.759} C_VEL
LIN {X 0,Y 208.814,Z 460.959,A -85,B 0,C 180,E1 -20987.633,E2 -20987.633} C_VEL
LIN {X 0,Y 211.563,Z 454.153,A -85,B 0,C 180,E1 -20990.923,E2 -20990.923} C_VEL
LIN {X 0,Y 214.409,Z 446.786,A -85,B 0,C 180,E1 -20993.674,E2 -20993.674} C_VEL
LIN {X 0,Y 217.777,Z 437.679,A -85,B 0,C 180,E1 -20996.342,E2 -20996.342} C_VEL
LIN {X 0,Y 221.446,Z 427.178,A -85,B 0,C 180,E1 -20998.687,E2 -20998.687} C_VEL
LIN {X 0,Y 224.284,Z 417.845,A -85,B 0,C 180,E1 -21000.35,E2 -21000.35} C_VEL
LIN {X 0,Y 227.364,Z 406.347,A -85,B 0,C 180,E1 -21001.961,E2 -21001.961} C_VEL
LIN {X 0,Y 229.965,Z 394.239,A -85,B 0,C 180,E1 -21003.243,E2 -21003.243} C_VEL
LIN {X 0,Y 232.231,Z 380.916,A -85,B 0,C 180,E1 -21004.243,E2 -21004.243} C_VEL
LIN {X 0,Y 233.71,Z 367.654,A -85,B 0,C 180,E1 -21004.902,E2 -21004.902} C_VEL
LIN {X 0,Y 236.406,Z 318.78,A -85,B 0,C 180,E1 -21006.435,E2 -21006.435} C_VEL
LIN {X 0,Y 235.14,Z 308.546,A -85,B 0,C 180,E1 -21007.155,E2 -21007.155} C_VEL
LIN {X 0,Y 229.408,Z 295.032,A -85,B 0,C 180,E1 -21009.115,E2 -21009.115} C_VEL
LIN {X 0,Y 223.702,Z 283.673,A -85,B 0,C 180,E1 -21011.161,E2 -21011.161} C_VEL
LIN {X 0,Y 218.545,Z 274.822,A -85,B 0,C 180,E1 -21013.13,E2 -21013.13} C_VEL
LIN {X 0,Y 215.321,Z 269.69,A -85,B 0,C 180,E1 -21014.439,E2 -21014.439} C_VEL
LIN {X 0,Y 211.677,Z 264.153,A -85,B 0,C 180,E1 -21016.031,E2 -21016.031} C_VEL
LIN {X 0,Y 208.59,Z 259.553,A -85,B 0,C 180,E1 -21017.471,E2 -21017.471} C_VEL
LIN {X 0,Y 208.309,Z 258.843,A -85,B 0,C 180,E1 -21017.761,E2 -21017.761} C_VEL
LIN {X 0,Y 206.679,Z 253.733,A -85,B 0,C 180,E1 -21021.836,E2 -21021.836} C_VEL
LIN {X 0,Y 206.7,Z 253.727,A -85,B 0,C 180,E1 -21024.689,E2 -21024.689} C_VEL
LIN {X 0,Y 206.714,Z 253.725,A -85,B 0,C 180,E1 -21029.338,E2 -21029.338} C_VEL
LIN {X 0,Y 206.734,Z 253.725,A -85,B 0,C 180,E1 -21033.772,E2 -21033.772} C_VEL
LIN {X 0,Y 206.758,Z 253.722,A -85,B 0,C 180,E1 -21038.043,E2 -21038.043} C_VEL
LIN {X 0,Y 206.874,Z 253.705,A -85,B 0,C 180,E1 -21042.197,E2 -21042.197} C_VEL
LIN {X 0,Y 206.914,Z 253.696,A -85,B 0,C 180,E1 -21046.246,E2 -21046.246} C_VEL
LIN {X 0,Y 207.106,Z 253.673,A -85,B 0,C 180,E1 -21050.231,E2 -21050.231} C_VEL
LIN {X 0,Y 207.168,Z 253.675,A -85,B 0,C 180,E1 -21052.201,E2 -21052.201} C_VEL
LIN {X 0,Y 207.383,Z 253.65,A -85,B 0,C 180,E1 -21058.058,E2 -21058.058} C_VEL
LIN {X 0,Y 207.512,Z 253.623,A -85,B 0,C 180,E1 -21060,E2 -21060} C_VEL
LIN {X 0,Y 207.382,Z 253.653,A -85,B 0,C 180,E1 -21061.942,E2 -21061.942} C_VEL
LIN {X 0,Y 207.169,Z 253.669,A -85,B 0,C 180,E1 -21067.799,E2 -21067.799} C_VEL
LIN {X 0,Y 206.948,Z 253.697,A -85,B 0,C 180,E1 -21071.757,E2 -21071.757} C_VEL
LIN {X 0,Y 206.888,Z 253.716,A -85,B 0,C 180,E1 -21076.91,E2 -21076.91} C_VEL
LIN {X 0,Y 207.927,Z 256.599,A -85,B 0,C 180,E1 -21077.534,E2 -21077.534} C_VEL
LIN {X 0,Y 209.879,Z 258.713,A -85,B 0,C 180,E1 -21078.423,E2 -21078.423} C_VEL
LIN {X 0,Y 210.719,Z 259.522,A -85,B 0,C 180,E1 -21078.788,E2 -21078.788} C_VEL
LIN {X 0,Y 212.643,Z 262.637,A -85,B 0,C 180,E1 -21079.676,E2 -21079.676} C_VEL
LIN {X 0,Y 214.476,Z 264.672,A -85,B 0,C 180,E1 -21080.438,E2 -21080.438} C_VEL
LIN {X 0,Y 217.174,Z 268.373,A -85,B 0,C 180,E1 -21081.537,E2 -21081.537} C_VEL
LIN {X 0,Y 221.853,Z 275.328,A -85,B 0,C 180,E1 -21083.34,E2 -21083.34} C_VEL
LIN {X 0,Y 227.513,Z 285.113,A -85,B 0,C 180,E1 -21085.379,E2 -21085.379} C_VEL
LIN {X 0,Y 233.149,Z 296.327,A -85,B 0,C 180,E1 -21087.303,E2 -21087.303} C_VEL
LIN {X 0,Y 237.075,Z 305.449,A -85,B 0,C 180,E1 -21088.585,E2 -21088.585} C_VEL
LIN {X 0,Y 233.891,Z 359.943,A -85,B 0,C 180,E1 -21090.29,E2 -21090.29} C_VEL
LIN {X 0,Y 232.394,Z 373.449,A -85,B 0,C 180,E1 -21091.04,E2 -21091.04} C_VEL
LIN {X 0,Y 230.254,Z 386.48,A -85,B 0,C 180,E1 -21092.112,E2 -21092.112} C_VEL
LIN {X 0,Y 227.637,Z 398.799,A -85,B 0,C 180,E1 -21093.531,E2 -21093.531} C_VEL
LIN {X 0,Y 224.72,Z 410.019,A -85,B 0,C 180,E1 -21095.215,E2 -21095.215} C_VEL
LIN {X 0,Y 221.806,Z 419.498,A -85,B 0,C 180,E1 -21097.015,E2 -21097.015} C_VEL
LIN {X 0,Y 218.36,Z 429.461,A -85,B 0,C 180,E1 -21099.426,E2 -21099.426} C_VEL
LIN {X 0,Y 215.159,Z 437.847,A -85,B 0,C 180,E1 -21102.003,E2 -21102.003} C_VEL
LIN {X 0,Y 212.317,Z 444.874,A -85,B 0,C 180,E1 -21104.764,E2 -21104.764} C_VEL
LIN {X 0,Y 209.664,Z 450.998,A -85,B 0,C 180,E1 -21107.902,E2 -21107.902} C_VEL
LIN {X 0,Y 207.546,Z 455.746,A -85,B 0,C 180,E1 -21111.154,E2 -21111.154} C_VEL
LIN {X 0,Y 205.987,Z 459.241,A -85,B 0,C 180,E1 -21114.548,E2 -21114.548} C_VEL
LIN {X 0,Y 205.202,Z 460.789,A -85,B 0,C 180,E1 -21116.771,E2 -21116.771} C_VEL
LIN {X 0,Y 204.567,Z 461.908,A -85,B 0,C 180,E1 -21119.192,E2 -21119.192} C_VEL
LIN {X 0,Y 204.213,Z 462.366,A -85,B 0,C 180,E1 -21121.196,E2 -21121.196} C_VEL
LIN {X 0,Y 203.995,Z 462.36,A -85,B 0,C 180,E1 -21123.605,E2 -21123.605} C_VEL
LIN {X 0,Y 203.95,Z 461.946,A -85,B 0,C 180,E1 -21125.574,E2 -21125.574} C_VEL
LIN {X 0,Y 204.123,Z 460.631,A -85,B 0,C 180,E1 -21128.376,E2 -21128.376} C_VEL
LIN {X 0,Y 204.76,Z 457.717,A -85,B 0,C 180,E1 -21132.006,E2 -21132.006} C_VEL
LIN {X 0,Y 205.58,Z 453.939,A -85,B 0,C 180,E1 -21135.143,E2 -21135.143} C_VEL
LIN {X 0,Y 206.722,Z 448.946,A -85,B 0,C 180,E1 -21138.23,E2 -21138.23} C_VEL
LIN {X 0,Y 208.306,Z 442.587,A -85,B 0,C 180,E1 -21141.267,E2 -21141.267} C_VEL
LIN {X 0,Y 210.381,Z 434.624,A -85,B 0,C 180,E1 -21144.248,E2 -21144.248} C_VEL
LIN {X 0,Y 212.44,Z 426.41,A -85,B 0,C 180,E1 -21146.681,E2 -21146.681} C_VEL
LIN {X 0,Y 214.772,Z 416.341,A -85,B 0,C 180,E1 -21149.062,E2 -21149.062} C_VEL
LIN {X 0,Y 217.041,Z 405.882,A -85,B 0,C 180,E1 -21151.02,E2 -21151.02} C_VEL
LIN {X 0,Y 219.239,Z 393.967,A -85,B 0,C 180,E1 -21152.756,E2 -21152.756} C_VEL
LIN {X 0,Y 221.044,Z 381.772,A -85,B 0,C 180,E1 -21154.102,E2 -21154.102} C_VEL
LIN {X 0,Y 222.487,Z 368.614,A -85,B 0,C 180,E1 -21155.153,E2 -21155.153} C_VEL
LIN {X 0,Y 223.477,Z 354.847,A -85,B 0,C 180,E1 -21155.84,E2 -21155.84} C_VEL
LIN {X 0,Y 226.061,Z 296.36,A -85,B 0,C 180,E1 -21157.704,E2 -21157.704} C_VEL
LIN {X 0,Y 221.353,Z 283.997,A -85,B 0,C 180,E1 -21158.839,E2 -21158.839} C_VEL
LIN {X 0,Y 214.015,Z 267.066,A -85,B 0,C 180,E1 -21160.623,E2 -21160.623} C_VEL
LIN {X 0,Y 208.35,Z 257.137,A -85,B 0,C 180,E1 -21161.978,E2 -21161.978} C_VEL
LIN {X 0,Y 207.075,Z 254.494,A -85,B 0,C 180,E1 -21162.314,E2 -21162.314} C_VEL
LIN {X 0,Y 206.931,Z 253.71,A -85,B 0,C 180,E1 -21162.442,E2 -21162.442} C_VEL
LIN {X 0,Y 206.875,Z 253.721,A -85,B 0,C 180,E1 -21167.803,E2 -21167.803} C_VEL
LIN {X 0,Y 206.748,Z 253.722,A -85,B 0,C 180,E1 -21173.391,E2 -21173.391} C_VEL
LIN {X 0,Y 206.69,Z 253.728,A -85,B 0,C 180,E1 -21178.426,E2 -21178.426} C_VEL
LIN {X 0,Y 206.696,Z 253.737,A -85,B 0,C 180,E1 -21182.958,E2 -21182.958} C_VEL
LIN {X 0,Y 206.68,Z 253.736,A -85,B 0,C 180,E1 -21187.739,E2 -21187.739} C_VEL
LIN {X 0,Y 206.641,Z 253.74,A -85,B 0,C 180,E1 -21191.562,E2 -21191.562} C_VEL
LIN {X 0,Y 206.631,Z 253.733,A -85,B 0,C 180,E1 -21195.582,E2 -21195.582} C_VEL
LIN {X 0,Y 206.66,Z 253.743,A -85,B 0,C 180,E1 -21199.748,E2 -21199.748} C_VEL
LIN {X 0,Y 206.698,Z 253.713,A -85,B 0,C 180,E1 -21204.688,E2 -21204.688} C_VEL
LIN {X 0,Y 206.706,Z 253.734,A -85,B 0,C 180,E1 -21209.336,E2 -21209.336} C_VEL
LIN {X 0,Y 206.732,Z 253.717,A -85,B 0,C 180,E1 -21213.772,E2 -21213.772} C_VEL
LIN {X 0,Y 206.756,Z 253.71,A -85,B 0,C 180,E1 -21218.043,E2 -21218.043} C_VEL
LIN {X 0,Y 206.873,Z 253.717,A -85,B 0,C 180,E1 -21222.196,E2 -21222.196} C_VEL
LIN {X 0,Y 206.912,Z 253.696,A -85,B 0,C 180,E1 -21226.245,E2 -21226.245} C_VEL
LIN {X 0,Y 207.131,Z 253.655,A -85,B 0,C 180,E1 -21230.232,E2 -21230.232} C_VEL
LIN {X 0,Y 207.187,Z 253.665,A -85,B 0,C 180,E1 -21232.202,E2 -21232.202} C_VEL
LIN {X 0,Y 207.381,Z 253.646,A -85,B 0,C 180,E1 -21238.058,E2 -21238.058} C_VEL
LIN {X 0,Y 207.513,Z 253.617,A -85,B 0,C 180,E1 -21240,E2 -21240} C_VEL
LIN {X 0,Y 207.381,Z 253.624,A -85,B 0,C 180,E1 -21241.942,E2 -21241.942} C_VEL
LIN {X 0,Y 207.187,Z 253.676,A -85,B 0,C 180,E1 -21247.798,E2 -21247.798} C_VEL
LIN {X 0,Y 206.974,Z 253.688,A -85,B 0,C 180,E1 -21251.755,E2 -21251.755} C_VEL
LIN {X 0,Y 206.865,Z 253.706,A -85,B 0,C 180,E1 -21255.771,E2 -21255.771} C_VEL
LIN {X 0,Y 206.782,Z 253.727,A -85,B 0,C 180,E1 -21259.869,E2 -21259.869} C_VEL
LIN {X 0,Y 206.762,Z 253.725,A -85,B 0,C 180,E1 -21264.072,E2 -21264.072} C_VEL
LIN {X 0,Y 206.743,Z 253.725,A -85,B 0,C 180,E1 -21268.419,E2 -21268.419} C_VEL
LIN {X 0,Y 206.701,Z 253.732,A -85,B 0,C 180,E1 -21272.957,E2 -21272.957} C_VEL
LIN {X 0,Y 206.678,Z 253.736,A -85,B 0,C 180,E1 -21277.74,E2 -21277.74} C_VEL
LIN {X 0,Y 206.639,Z 253.736,A -85,B 0,C 180,E1 -21281.563,E2 -21281.563} C_VEL
LIN {X 0,Y 206.632,Z 253.748,A -85,B 0,C 180,E1 -21285.582,E2 -21285.582} C_VEL
LIN {X 0,Y 206.704,Z 253.833,A -85,B 0,C 180,E1 -21289.03,E2 -21289.03} C_VEL
LIN {X 0,Y 208.616,Z 261.454,A -85,B 0,C 180,E1 -21292.869,E2 -21292.869} C_VEL
LIN {X 0,Y 213.023,Z 271.357,A -85,B 0,C 180,E1 -21294.002,E2 -21294.002} C_VEL
LIN {X 0,Y 214.688,Z 276.733,A -85,B 0,C 180,E1 -21294.485,E2 -21294.485} C_VEL
LIN {X 0,Y 215.868,Z 286.334,A -85,B 0,C 180,E1 -21295.054,E2 -21295.054} C_VEL
LIN {X 0,Y 216.32,Z 294.235,A -85,B 0,C 180,E1 -21295.438,E2 -21295.438} C_VEL
LIN {X 0,Y 217.293,Z 302.011,A -85,B 0,C 180,E1 -21295.89,E2 -21295.89} C_VEL
LIN {X 0,Y 219.116,Z 316.791,A -85,B 0,C 180,E1 -21296.728,E2 -21296.728} C_VEL
LIN {X 0,Y 216.679,Z 370.058,A -85,B 0,C 180,E1 -21298.514,E2 -21298.514} C_VEL
LIN {X 0,Y 215.373,Z 383.181,A -85,B 0,C 180,E1 -21299.277,E2 -21299.277} C_VEL
LIN {X 0,Y 213.604,Z 396.292,A -85,B 0,C 180,E1 -21300.428,E2 -21300.428} C_VEL
LIN {X 0,Y 211.591,Z 407.363,A -85,B 0,C 180,E1 -21301.751,E2 -21301.751} C_VEL
LIN {X 0,Y 209.159,Z 418.95,A -85,B 0,C 180,E1 -21303.563,E2 -21303.563} C_VEL
LIN {X 0,Y 206.728,Z 429.406,A -85,B 0,C 180,E1 -21305.657,E2 -21305.657} C_VEL
LIN {X 0,Y 204.619,Z 437.955,A -85,B 0,C 180,E1 -21307.802,E2 -21307.802} C_VEL
LIN {X 0,Y 202.746,Z 445.841,A -85,B 0,C 180,E1 -21310.247,E2 -21310.247} C_VEL
LIN {X 0,Y 200.663,Z 453.502,A -85,B 0,C 180,E1 -21313.206,E2 -21313.206} C_VEL
LIN {X 0,Y 198.858,Z 460.568,A -85,B 0,C 180,E1 -21316.72,E2 -21316.72} C_VEL
LIN {X 0,Y 197.967,Z 465.239,A -85,B 0,C 180,E1 -21319.776,E2 -21319.776} C_VEL
LIN {X 0,Y 197.587,Z 467.697,A -85,B 0,C 180,E1 -21321.821,E2 -21321.821} C_VEL
LIN {X 0,Y 197.343,Z 469.693,A -85,B 0,C 180,E1 -21323.867,E2 -21323.867} C_VEL
LIN {X 0,Y 197.244,Z 471.389,A -85,B 0,C 180,E1 -21326.088,E2 -21326.088} C_VEL
LIN {X 0,Y 197.269,Z 472.405,A -85,B 0,C 180,E1 -21327.959,E2 -21327.959} C_VEL
LIN {X 0,Y 197.379,Z 473.103,A -85,B 0,C 180,E1 -21330,E2 -21330} C_VEL
LIN {X 0,Y 197.243,Z 473.328,A -85,B 0,C 180,E1 -21333.909,E2 -21333.909} C_VEL
LIN {X 0,Y 197.341,Z 472.822,A -85,B 0,C 180,E1 -21336.133,E2 -21336.133} C_VEL
LIN {X 0,Y 198.039,Z 470.6,A -85,B 0,C 180,E1 -21340.221,E2 -21340.221} C_VEL
LIN {X 0,Y 199.086,Z 467.863,A -85,B 0,C 180,E1 -21343.265,E2 -21343.265} C_VEL
LIN {X 0,Y 200.618,Z 464.125,A -85,B 0,C 180,E1 -21346.276,E2 -21346.276} C_VEL
LIN {X 0,Y 202.855,Z 459.288,A -85,B 0,C 180,E1 -21349.216,E2 -21349.216} C_VEL
LIN {X 0,Y 205.443,Z 453.214,A -85,B 0,C 180,E1 -21352.105,E2 -21352.105} C_VEL
LIN {X 0,Y 208.46,Z 445.711,A -85,B 0,C 180,E1 -21354.925,E2 -21354.925} C_VEL
LIN {X 0,Y 211.447,Z 438.083,A -85,B 0,C 180,E1 -21357.195,E2 -21357.195} C_VEL
LIN {X 0,Y 214.872,Z 428.85,A -85,B 0,C 180,E1 -21359.381,E2 -21359.381} C_VEL
LIN {X 0,Y 218.214,Z 418.624,A -85,B 0,C 180,E1 -21361.288,E2 -21361.288} C_VEL
LIN {X 0,Y 221.421,Z 407.34,A -85,B 0,C 180,E1 -21362.926,E2 -21362.926} C_VEL
LIN {X 0,Y 224.146,Z 395.681,A -85,B 0,C 180,E1 -21364.224,E2 -21364.224} C_VEL
LIN {X 0,Y 226.449,Z 382.979,A -85,B 0,C 180,E1 -21365.245,E2 -21365.245} C_VEL
LIN {X 0,Y 228.172,Z 369.558,A -85,B 0,C 180,E1 -21365.964,E2 -21365.964} C_VEL
LIN {X 0,Y 231.127,Z 319.98,A -85,B 0,C 180,E1 -21367.561,E2 -21367.561} C_VEL
LIN {X 0,Y 230.055,Z 311.295,A -85,B 0,C 180,E1 -21368.205,E2 -21368.205} C_VEL
LIN {X 0,Y 224.327,Z 297.732,A -85,B 0,C 180,E1 -21370.3,E2 -21370.3} C_VEL
LIN {X 0,Y 218.75,Z 286.618,A -85,B 0,C 180,E1 -21372.443,E2 -21372.443} C_VEL
LIN {X 0,Y 212.45,Z 275.78,A -85,B 0,C 180,E1 -21375.063,E2 -21375.063} C_VEL
LIN {X 0,Y 208.291,Z 269.47,A -85,B 0,C 180,E1 -21376.96,E2 -21376.96} C_VEL
LIN {X 0,Y 204.772,Z 264.23,A -85,B 0,C 180,E1 -21378.699,E2 -21378.699} C_VEL
LIN {X 0,Y 201.71,Z 260.069,A -85,B 0,C 180,E1 -21380.33,E2 -21380.33} C_VEL
LIN {X 0,Y 200.923,Z 258.584,A -85,B 0,C 180,E1 -21380.868,E2 -21380.868} C_VEL
LIN {X 0,Y 199.643,Z 254.606,A -85,B 0,C 180,E1 -21384.563,E2 -21384.563} C_VEL
LIN {X 0,Y 199.694,Z 254.599,A -85,B 0,C 180,E1 -21388.136,E2 -21388.136} C_VEL
LIN {X 0,Y 199.687,Z 254.598,A -85,B 0,C 180,E1 -21392.772,E2 -21392.772} C_VEL
LIN {X 0,Y 199.739,Z 254.592,A -85,B 0,C 180,E1 -21397.229,E2 -21397.229} C_VEL
LIN {X 0,Y 199.797,Z 254.584,A -85,B 0,C 180,E1 -21401.758,E2 -21401.758} C_VEL
LIN {X 0,Y 199.849,Z 254.576,A -85,B 0,C 180,E1 -21405.749,E2 -21405.749} C_VEL
LIN {X 0,Y 200.071,Z 254.55,A -85,B 0,C 180,E1 -21409.884,E2 -21409.884} C_VEL
LIN {X 0,Y 200.034,Z 254.559,A -85,B 0,C 180,E1 -21413.95,E2 -21413.95} C_VEL
LIN {X 0,Y 200.322,Z 254.53,A -85,B 0,C 180,E1 -21417.99,E2 -21417.99} C_VEL
LIN {X 0,Y 200.477,Z 254.499,A -85,B 0,C 180,E1 -21420,E2 -21420} C_VEL
LIN {X 0,Y 200.03,Z 254.556,A -85,B 0,C 180,E1 -21424.03,E2 -21424.03} C_VEL
LIN {X 0,Y 200.112,Z 254.547,A -85,B 0,C 180,E1 -21428.076,E2 -21428.076} C_VEL
LIN {X 0,Y 199.892,Z 254.577,A -85,B 0,C 180,E1 -21432.178,E2 -21432.178} C_VEL
LIN {X 0,Y 199.899,Z 254.724,A -85,B 0,C 180,E1 -21433.858,E2 -21433.858} C_VEL
LIN {X 0,Y 200.627,Z 257.056,A -85,B 0,C 180,E1 -21434.389,E2 -21434.389} C_VEL
LIN {X 0,Y 202.365,Z 259.209,A -85,B 0,C 180,E1 -21435.356,E2 -21435.356} C_VEL
LIN {X 0,Y 203.946,Z 260.289,A -85,B 0,C 180,E1 -21436.137,E2 -21436.137} C_VEL
LIN {X 0,Y 205.863,Z 263.578,A -85,B 0,C 180,E1 -21437.158,E2 -21437.158} C_VEL
LIN {X 0,Y 207.767,Z 265.576,A -85,B 0,C 180,E1 -21438.043,E2 -21438.043} C_VEL
LIN {X 0,Y 210.263,Z 269.154,A -85,B 0,C 180,E1 -21439.21,E2 -21439.21} C_VEL
LIN {X 0,Y 211.793,Z 271.196,A -85,B 0,C 180,E1 -21439.885,E2 -21439.885} C_VEL
LIN {X 0,Y 217.529,Z 279.451,A -85,B 0,C 180,E1 -21442.248,E2 -21442.248} C_VEL
LIN {X 0,Y 222.077,Z 287.331,A -85,B 0,C 180,E1 -21444.021,E2 -21444.021} C_VEL
LIN {X 0,Y 227.913,Z 298.736,A -85,B 0,C 180,E1 -21446.129,E2 -21446.129} C_VEL
LIN {X 0,Y 231.741,Z 307.722,A -85,B 0,C 180,E1 -21447.483,E2 -21447.483} C_VEL
LIN {X 0,Y 228.471,Z 360.568,A -85,B 0,C 180,E1 -21449.163,E2 -21449.163} C_VEL
LIN {X 0,Y 226.853,Z 374.328,A -85,B 0,C 180,E1 -21449.948,E2 -21449.948} C_VEL
LIN {X 0,Y 224.826,Z 386.204,A -85,B 0,C 180,E1 -21450.942,E2 -21450.942} C_VEL
LIN {X 0,Y 222.252,Z 398.024,A -85,B 0,C 180,E1 -21452.302,E2 -21452.302} C_VEL
LIN {X 0,Y 219.24,Z 409.141,A -85,B 0,C 180,E1 -21453.957,E2 -21453.957} C_VEL
LIN {X 0,Y 216.12,Z 419.013,A -85,B 0,C 180,E1 -21455.827,E2 -21455.827} C_VEL
LIN {X 0,Y 212.673,Z 428.617,A -85,B 0,C 180,E1 -21458.143,E2 -21458.143} C_VEL
LIN {X 0,Y 209.121,Z 437.459,A -85,B 0,C 180,E1 -21460.873,E2 -21460.873} C_VEL
LIN {X 0,Y 206.312,Z 444.028,A -85,B 0,C 180,E1 -21463.453,E2 -21463.453} C_VEL
LIN {X 0,Y 203.575,Z 450.075,A -85,B 0,C 180,E1 -21466.468,E2 -21466.468} C_VEL
LIN {X 0,Y 201.368,Z 454.791,A -85,B 0,C 180,E1 -21469.559,E2 -21469.559} C_VEL
LIN {X 0,Y 199.423,Z 458.745,A -85,B 0,C 180,E1 -21473.194,E2 -21473.194} C_VEL
LIN {X 0,Y 198.526,Z 460.517,A -85,B 0,C 180,E1 -21475.499,E2 -21475.499} C_VEL
LIN {X 0,Y 197.587,Z 462.037,A -85,B 0,C 180,E1 -21478.613,E2 -21478.613} C_VEL
LIN {X 0,Y 196.976,Z 462.651,A -85,B 0,C 180,E1 -21482.365,E2 -21482.365} C_VEL
LIN {X 0,Y 196.847,Z 462.342,A -85,B 0,C 180,E1 -21484.632,E2 -21484.632} C_VEL
LIN {X 0,Y 196.983,Z 460.974,A -85,B 0,C 180,E1 -21488.07,E2 -21488.07} C_VEL
LIN {X 0,Y 197.753,Z 457.569,A -85,B 0,C 180,E1 -21492.418,E2 -21492.418} C_VEL
LIN {X 0,Y 198.625,Z 453.676,A -85,B 0,C 180,E1 -21495.659,E2 -21495.659} C_VEL
LIN {X 0,Y 199.824,Z 448.744,A -85,B 0,C 180,E1 -21498.748,E2 -21498.748} C_VEL
LIN {X 0,Y 201.56,Z 442.07,A -85,B 0,C 180,E1 -21501.982,E2 -21501.982} C_VEL
LIN {X 0,Y 203.354,Z 435.4,A -85,B 0,C 180,E1 -21504.543,E2 -21504.543} C_VEL
LIN {X 0,Y 205.495,Z 427.32,A -85,B 0,C 180,E1 -21507.059,E2 -21507.059} C_VEL
LIN {X 0,Y 207.867,Z 417.424,A -85,B 0,C 180,E1 -21509.515,E2 -21509.515} C_VEL
LIN {X 0,Y 210.385,Z 406.332,A -85,B 0,C 180,E1 -21511.675,E2 -21511.675} C_VEL
LIN {X 0,Y 212.513,Z 395.264,A -85,B 0,C 180,E1 -21513.363,E2 -21513.363} C_VEL
LIN {X 0,Y 214.518,Z 382.619,A -85,B 0,C 180,E1 -21514.815,E2 -21514.815} C_VEL
LIN {X 0,Y 215.971,Z 369.854,A -85,B 0,C 180,E1 -21515.89,E2 -21515.89} C_VEL
LIN {X 0,Y 217.059,Z 356.473,A -85,B 0,C 180,E1 -21516.606,E2 -21516.606} C_VEL
LIN {X 0,Y 219.755,Z 298.094,A -85,B 0,C 180,E1 -21518.521,E2 -21518.521} C_VEL
LIN {X 0,Y 215.519,Z 287.005,A -85,B 0,C 180,E1 -21519.583,E2 -21519.583} C_VEL
LIN {X 0,Y 208.68,Z 270.955,A -85,B 0,C 180,E1 -21521.337,E2 -21521.337} C_VEL
LIN {X 0,Y 201.264,Z 257.985,A -85,B 0,C 180,E1 -21523.199,E2 -21523.199} C_VEL
LIN {X 0,Y 200.029,Z 255.444,A -85,B 0,C 180,E1 -21523.541,E2 -21523.541} C_VEL
LIN {X 0,Y 199.865,Z 254.592,A -85,B 0,C 180,E1 -21523.682,E2 -21523.682} C_VEL
LIN {X 0,Y 199.785,Z 254.603,A -85,B 0,C 180,E1 -21528.457,E2 -21528.457} C_VEL
LIN {X 0,Y 199.71,Z 254.6,A -85,B 0,C 180,E1 -21533.798,E2 -21533.798} C_VEL
LIN {X 0,Y 199.666,Z 254.602,A -85,B 0,C 180,E1 -21538.361,E2 -21538.361} C_VEL
LIN {X 0,Y 199.666,Z 254.614,A -85,B 0,C 180,E1 -21542.352,E2 -21542.352} C_VEL
LIN {X 0,Y 199.624,Z 254.61,A -85,B 0,C 180,E1 -21546.762,E2 -21546.762} C_VEL
LIN {X 0,Y 199.608,Z 254.621,A -85,B 0,C 180,E1 -21549.327,E2 -21549.327} C_VEL
LIN {X 0,Y 199.572,Z 254.614,A -85,B 0,C 180,E1 -21552.309,E2 -21552.309} C_VEL
LIN {X 0,Y 199.577,Z 254.61,A -85,B 0,C 180,E1 -21555.227,E2 -21555.227} C_VEL
LIN {X 0,Y 199.579,Z 254.624,A -85,B 0,C 180,E1 -21558.004,E2 -21558.004} C_VEL
LIN {X 0,Y 199.61,Z 254.616,A -85,B 0,C 180,E1 -21560.767,E2 -21560.767} C_VEL
LIN {X 0,Y 199.611,Z 254.599,A -85,B 0,C 180,E1 -21565.713,E2 -21565.713} C_VEL
LIN {X 0,Y 199.692,Z 254.606,A -85,B 0,C 180,E1 -21568.135,E2 -21568.135} C_VEL
LIN {X 0,Y 199.685,Z 254.602,A -85,B 0,C 180,E1 -21572.771,E2 -21572.771} C_VEL
LIN {X 0,Y 199.737,Z 254.578,A -85,B 0,C 180,E1 -21577.229,E2 -21577.229} C_VEL
LIN {X 0,Y 199.796,Z 254.596,A -85,B 0,C 180,E1 -21581.757,E2 -21581.757} C_VEL
LIN {X 0,Y 199.847,Z 254.579,A -85,B 0,C 180,E1 -21585.749,E2 -21585.749} C_VEL
LIN {X 0,Y 200.074,Z 254.53,A -85,B 0,C 180,E1 -21589.884,E2 -21589.884} C_VEL
LIN {X 0,Y 200.131,Z 254.541,A -85,B 0,C 180,E1 -21591.925,E2 -21591.925} C_VEL
LIN {X 0,Y 200.321,Z 254.526,A -85,B 0,C 180,E1 -21597.989,E2 -21597.989} C_VEL
LIN {X 0,Y 200.478,Z 254.492,A -85,B 0,C 180,E1 -21600,E2 -21600} C_VEL
LIN {X 0,Y 200.03,Z 254.55,A -85,B 0,C 180,E1 -21604.029,E2 -21604.029} C_VEL
LIN {X 0,Y 200.131,Z 254.557,A -85,B 0,C 180,E1 -21608.075,E2 -21608.075} C_VEL
LIN {X 0,Y 199.905,Z 254.563,A -85,B 0,C 180,E1 -21612.177,E2 -21612.177} C_VEL
LIN {X 0,Y 199.803,Z 254.589,A -85,B 0,C 180,E1 -21616.343,E2 -21616.343} C_VEL
LIN {X 0,Y 199.699,Z 254.604,A -85,B 0,C 180,E1 -21620.605,E2 -21620.605} C_VEL
LIN {X 0,Y 199.672,Z 254.612,A -85,B 0,C 180,E1 -21624.984,E2 -21624.984} C_VEL
LIN {X 0,Y 199.674,Z 254.607,A -85,B 0,C 180,E1 -21629.522,E2 -21629.522} C_VEL
LIN {X 0,Y 199.676,Z 254.61,A -85,B 0,C 180,E1 -21632.359,E2 -21632.359} C_VEL
LIN {X 0,Y 199.622,Z 254.617,A -85,B 0,C 180,E1 -21636.763,E2 -21636.763} C_VEL
LIN {X 0,Y 199.607,Z 254.621,A -85,B 0,C 180,E1 -21639.328,E2 -21639.328} C_VEL
LIN {X 0,Y 199.571,Z 254.611,A -85,B 0,C 180,E1 -21642.31,E2 -21642.31} C_VEL
LIN {X 0,Y 199.578,Z 254.627,A -85,B 0,C 180,E1 -21645.229,E2 -21645.229} C_VEL
LIN {X 0,Y 199.614,Z 254.676,A -85,B 0,C 180,E1 -21648.093,E2 -21648.093} C_VEL
LIN {X 0,Y 201.355,Z 261.356,A -85,B 0,C 180,E1 -21651.583,E2 -21651.583} C_VEL
LIN {X 0,Y 208.726,Z 277.617,A -85,B 0,C 180,E1 -21653.565,E2 -21653.565} C_VEL
LIN {X 0,Y 215.824,Z 295.426,A -85,B 0,C 180,E1 -21655.411,E2 -21655.411} C_VEL
LIN {X 0,Y 216.884,Z 299.282,A -85,B 0,C 180,E1 -21655.722,E2 -21655.722} C_VEL
LIN {X 0,Y 217.293,Z 302.011,A -85,B 0,C 180,E1 -21655.89,E2 -21655.89} C_VEL
LIN {X 0,Y 217.662,Z 305.834,A -85,B 0,C 180,E1 -21656.094,E2 -21656.094} C_VEL
LIN {X 0,Y 217.099,Z 311.697,A -85,B 0,C 180,E1 -21656.244,E2 -21656.244} C_VEL
LIN {X 0,Y 212.689,Z 329.335,A -85,B 0,C 180,E1 -21656.306,E2 -21656.306} C_VEL
LIN {X 0,Y 212.222,Z 333.343,A -85,B 0,C 180,E1 -21656.398,E2 -21656.398} C_VEL
LIN {X 0,Y 210.315,Z 370.334,A -85,B 0,C 180,E1 -21657.679,E2 -21657.679} C_VEL
LIN {X 0,Y 208.902,Z 383.839,A -85,B 0,C 180,E1 -21658.5,E2 -21658.5} C_VEL
LIN {X 0,Y 207.054,Z 396.664,A -85,B 0,C 180,E1 -21659.676,E2 -21659.676} C_VEL
LIN {X 0,Y 205.003,Z 407.617,A -85,B 0,C 180,E1 -21661.038,E2 -21661.038} C_VEL
LIN {X 0,Y 202.485,Z 419.123,A -85,B 0,C 180,E1 -21662.9,E2 -21662.9} C_VEL
LIN {X 0,Y 199.973,Z 429.514,A -85,B 0,C 180,E1 -21665.056,E2 -21665.056} C_VEL
LIN {X 0,Y 197.643,Z 438.6,A -85,B 0,C 180,E1 -21667.447,E2 -21667.447} C_VEL
LIN {X 0,Y 195.626,Z 446.527,A -85,B 0,C 180,E1 -21670.045,E2 -21670.045} C_VEL
LIN {X 0,Y 193.521,Z 454.033,A -85,B 0,C 180,E1 -21673.111,E2 -21673.111} C_VEL
LIN {X 0,Y 191.918,Z 460.046,A -85,B 0,C 180,E1 -21676.23,E2 -21676.23} C_VEL
LIN {X 0,Y 190.959,Z 464.788,A -85,B 0,C 180,E1 -21679.397,E2 -21679.397} C_VEL
LIN {X 0,Y 190.364,Z 468.383,A -85,B 0,C 180,E1 -21682.576,E2 -21682.576} C_VEL
LIN {X 0,Y 190.138,Z 471.333,A -85,B 0,C 180,E1 -21686.367,E2 -21686.367} C_VEL
LIN {X 0,Y 190.281,Z 472.863,A -85,B 0,C 180,E1 -21690,E2 -21690} C_VEL
LIN {X 0,Y 190.134,Z 473.185,A -85,B 0,C 180,E1 -21693.614,E2 -21693.614} C_VEL
LIN {X 0,Y 190.279,Z 472.68,A -85,B 0,C 180,E1 -21696.362,E2 -21696.362} C_VEL
LIN {X 0,Y 191.033,Z 470.527,A -85,B 0,C 180,E1 -21700.6,E2 -21700.6} C_VEL
LIN {X 0,Y 192.162,Z 467.848,A -85,B 0,C 180,E1 -21703.753,E2 -21703.753} C_VEL
LIN {X 0,Y 193.812,Z 464.179,A -85,B 0,C 180,E1 -21706.864,E2 -21706.864} C_VEL
LIN {X 0,Y 196.161,Z 459.422,A -85,B 0,C 180,E1 -21709.899,E2 -21709.899} C_VEL
LIN {X 0,Y 198.889,Z 453.442,A -85,B 0,C 180,E1 -21712.874,E2 -21712.874} C_VEL
LIN {X 0,Y 202.065,Z 446.031,A -85,B 0,C 180,E1 -21715.77,E2 -21715.77} C_VEL
LIN {X 0,Y 205.182,Z 438.505,A -85,B 0,C 180,E1 -21718.097,E2 -21718.097} C_VEL
LIN {X 0,Y 208.751,Z 429.42,A -85,B 0,C 180,E1 -21720.332,E2 -21720.332} C_VEL
LIN {X 0,Y 212.216,Z 419.402,A -85,B 0,C 180,E1 -21722.277,E2 -21722.277} C_VEL
LIN {X 0,Y 215.558,Z 408.33,A -85,B 0,C 180,E1 -21723.941,E2 -21723.941} C_VEL
LIN {X 0,Y 218.592,Z 396.012,A -85,B 0,C 180,E1 -21725.361,E2 -21725.361} C_VEL
LIN {X 0,Y 221.001,Z 383.619,A -85,B 0,C 180,E1 -21726.39,E2 -21726.39} C_VEL
LIN {X 0,Y 222.879,Z 369.653,A -85,B 0,C 180,E1 -21727.165,E2 -21727.165} C_VEL
LIN {X 0,Y 225.197,Z 333.67,A -85,B 0,C 180,E1 -21728.358,E2 -21728.358} C_VEL
LIN {X 0,Y 225.902,Z 319.957,A -85,B 0,C 180,E1 -21728.826,E2 -21728.826} C_VEL
LIN {X 0,Y 225.174,Z 314.439,A -85,B 0,C 180,E1 -21729.271,E2 -21729.271} C_VEL
LIN {X 0,Y 220.299,Z 302.557,A -85,B 0,C 180,E1 -21731.161,E2 -21731.161} C_VEL
LIN {X 0,Y 214.564,Z 290.687,A -85,B 0,C 180,E1 -21733.524,E2 -21733.524} C_VEL
LIN {X 0,Y 208.588,Z 280.47,A -85,B 0,C 180,E1 -21736.168,E2 -21736.168} C_VEL
LIN {X 0,Y 204.995,Z 274.797,A -85,B 0,C 180,E1 -21737.914,E2 -21737.914} C_VEL
LIN {X 0,Y 201.878,Z 270.036,A -85,B 0,C 180,E1 -21739.546,E2 -21739.546} C_VEL
LIN {X 0,Y 198.59,Z 265.207,A -85,B 0,C 180,E1 -21741.436,E2 -21741.436} C_VEL
LIN {X 0,Y 194.363,Z 259.886,A -85,B 0,C 180,E1 -21744.091,E2 -21744.091} C_VEL
LIN {X 0,Y 193.51,Z 258.135,A -85,B 0,C 180,E1 -21744.791,E2 -21744.791} C_VEL
LIN {X 0,Y 192.646,Z 255.478,A -85,B 0,C 180,E1 -21747.86,E2 -21747.86} C_VEL
LIN {X 0,Y 192.665,Z 255.476,A -85,B 0,C 180,E1 -21751.692,E2 -21751.692} C_VEL
LIN {X 0,Y 192.707,Z 255.469,A -85,B 0,C 180,E1 -21756.349,E2 -21756.349} C_VEL
LIN {X 0,Y 192.733,Z 255.463,A -85,B 0,C 180,E1 -21761.458,E2 -21761.458} C_VEL
LIN {X 0,Y 192.773,Z 255.459,A -85,B 0,C 180,E1 -21765.215,E2 -21765.215} C_VEL
LIN {X 0,Y 192.982,Z 255.435,A -85,B 0,C 180,E1 -21769.509,E2 -21769.509} C_VEL
LIN {X 0,Y 193.062,Z 255.425,A -85,B 0,C 180,E1 -21771.627,E2 -21771.627} C_VEL
LIN {X 0,Y 193.264,Z 255.409,A -85,B 0,C 180,E1 -21777.916,E2 -21777.916} C_VEL
LIN {X 0,Y 193.441,Z 255.376,A -85,B 0,C 180,E1 -21780,E2 -21780} C_VEL
LIN {X 0,Y 192.976,Z 255.434,A -85,B 0,C 180,E1 -21784.177,E2 -21784.177} C_VEL
LIN {X 0,Y 193.028,Z 255.436,A -85,B 0,C 180,E1 -21789.43,E2 -21789.43} C_VEL
LIN {X 0,Y 193.005,Z 255.449,A -85,B 0,C 180,E1 -21790.183,E2 -21790.183} C_VEL
LIN {X 0,Y 193.673,Z 257.838,A -85,B 0,C 180,E1 -21790.795,E2 -21790.795} C_VEL
LIN {X 0,Y 195.372,Z 260.044,A -85,B 0,C 180,E1 -21791.938,E2 -21791.938} C_VEL
LIN {X 0,Y 197.188,Z 261.282,A -85,B 0,C 180,E1 -21793.002,E2 -21793.002} C_VEL
LIN {X 0,Y 198.931,Z 264.414,A -85,B 0,C 180,E1 -21794.122,E2 -21794.122} C_VEL
LIN {X 0,Y 201.457,Z 266.922,A -85,B 0,C 180,E1 -21795.492,E2 -21795.492} C_VEL
LIN {X 0,Y 203.847,Z 270.39,A -85,B 0,C 180,E1 -21796.778,E2 -21796.778} C_VEL
LIN {X 0,Y 205.169,Z 272.094,A -85,B 0,C 180,E1 -21797.432,E2 -21797.432} C_VEL
LIN {X 0,Y 208.592,Z 276.765,A -85,B 0,C 180,E1 -21799.055,E2 -21799.055} C_VEL
LIN {X 0,Y 214.513,Z 285.6,A -85,B 0,C 180,E1 -21801.628,E2 -21801.628} C_VEL
LIN {X 0,Y 219.95,Z 295.531,A -85,B 0,C 180,E1 -21803.827,E2 -21803.827} C_VEL
LIN {X 0,Y 224.755,Z 305.782,A -85,B 0,C 180,E1 -21805.651,E2 -21805.651} C_VEL
LIN {X 0,Y 226.511,Z 310.252,A -85,B 0,C 180,E1 -21806.316,E2 -21806.316} C_VEL
LIN {X 0,Y 223.292,Z 360.261,A -85,B 0,C 180,E1 -21807.932,E2 -21807.932} C_VEL
LIN {X 0,Y 221.693,Z 373.583,A -85,B 0,C 180,E1 -21808.689,E2 -21808.689} C_VEL
LIN {X 0,Y 219.501,Z 385.977,A -85,B 0,C 180,E1 -21809.717,E2 -21809.717} C_VEL
LIN {X 0,Y 216.738,Z 398.102,A -85,B 0,C 180,E1 -21811.121,E2 -21811.121} C_VEL
LIN {X 0,Y 213.435,Z 409.771,A -85,B 0,C 180,E1 -21812.895,E2 -21812.895} C_VEL
LIN {X 0,Y 210.24,Z 419.376,A -85,B 0,C 180,E1 -21814.758,E2 -21814.758} C_VEL
LIN {X 0,Y 206.783,Z 428.515,A -85,B 0,C 180,E1 -21816.995,E2 -21816.995} C_VEL
LIN {X 0,Y 203.174,Z 437.105,A -85,B 0,C 180,E1 -21819.678,E2 -21819.678} C_VEL
LIN {X 0,Y 200.007,Z 444.073,A -85,B 0,C 180,E1 -21822.446,E2 -21822.446} C_VEL
LIN {X 0,Y 197.166,Z 450.013,A -85,B 0,C 180,E1 -21825.472,E2 -21825.472} C_VEL
LIN {X 0,Y 195.074,Z 454.17,A -85,B 0,C 180,E1 -21828.202,E2 -21828.202} C_VEL
LIN {X 0,Y 192.972,Z 458.22,A -85,B 0,C 180,E1 -21831.747,E2 -21831.747} C_VEL
LIN {X 0,Y 191.891,Z 460.156,A -85,B 0,C 180,E1 -21834.126,E2 -21834.126} C_VEL
LIN {X 0,Y 190.655,Z 462.16,A -85,B 0,C 180,E1 -21837.978,E2 -21837.978} C_VEL
LIN {X 0,Y 189.991,Z 462.812,A -85,B 0,C 180,E1 -21841.257,E2 -21841.257} C_VEL
LIN {X 0,Y 189.801,Z 462.716,A -85,B 0,C 180,E1 -21843.619,E2 -21843.619} C_VEL
LIN {X 0,Y 189.86,Z 461.317,A -85,B 0,C 180,E1 -21847.733,E2 -21847.733} C_VEL
LIN {X 0,Y 190.47,Z 458.502,A -85,B 0,C 180,E1 -21851.721,E2 -21851.721} C_VEL
LIN {X 0,Y 191.347,Z 454.879,A -85,B 0,C 180,E1 -21855.102,E2 -21855.102} C_VEL
LIN {X 0,Y 192.584,Z 449.887,A -85,B 0,C 180,E1 -21858.528,E2 -21858.528} C_VEL
LIN {X 0,Y 194.165,Z 443.894,A -85,B 0,C 180,E1 -21861.675,E2 -21861.675} C_VEL
LIN {X 0,Y 196.354,Z 436.119,A -85,B 0,C 180,E1 -21864.866,E2 -21864.866} C_VEL
LIN {X 0,Y 198.547,Z 428.157,A -85,B 0,C 180,E1 -21867.464,E2 -21867.464} C_VEL
LIN {X 0,Y 200.999,Z 418.452,A -85,B 0,C 180,E1 -21870,E2 -21870} C_VEL
LIN {X 0,Y 203.641,Z 407.288,A -85,B 0,C 180,E1 -21872.269,E2 -21872.269} C_VEL
LIN {X 0,Y 206.061,Z 395.332,A -85,B 0,C 180,E1 -21874.156,E2 -21874.156} C_VEL
LIN {X 0,Y 208.021,Z 383.382,A -85,B 0,C 180,E1 -21875.574,E2 -21875.574} C_VEL
LIN {X 0,Y 209.633,Z 369.961,A -85,B 0,C 180,E1 -21876.738,E2 -21876.738} C_VEL
LIN {X 0,Y 210.682,Z 357.697,A -85,B 0,C 180,E1 -21877.427,E2 -21877.427} C_VEL
LIN {X 0,Y 213.48,Z 299.66,A -85,B 0,C 180,E1 -21879.384,E2 -21879.384} C_VEL
LIN {X 0,Y 209.587,Z 289.595,A -85,B 0,C 180,E1 -21880.408,E2 -21880.408} C_VEL
LIN {X 0,Y 203.295,Z 274.698,A -85,B 0,C 180,E1 -21882.1,E2 -21882.1} C_VEL
LIN {X 0,Y 194.305,Z 259.035,A -85,B 0,C 180,E1 -21884.478,E2 -21884.478} C_VEL
LIN {X 0,Y 192.995,Z 256.576,A -85,B 0,C 180,E1 -21884.856,E2 -21884.856} C_VEL
LIN {X 0,Y 192.775,Z 255.478,A -85,B 0,C 180,E1 -21884.988,E2 -21884.988} C_VEL
LIN {X 0,Y 192.693,Z 255.487,A -85,B 0,C 180,E1 -21889.162,E2 -21889.162} C_VEL
LIN {X 0,Y 192.642,Z 255.484,A -85,B 0,C 180,E1 -21894.208,E2 -21894.208} C_VEL
LIN {X 0,Y 192.603,Z 255.482,A -85,B 0,C 180,E1 -21898.865,E2 -21898.865} C_VEL
LIN {X 0,Y 192.595,Z 255.493,A -85,B 0,C 180,E1 -21903.186,E2 -21903.186} C_VEL
LIN {X 0,Y 192.552,Z 255.5,A -85,B 0,C 180,E1 -21908.351,E2 -21908.351} C_VEL
LIN {X 0,Y 192.489,Z 255.49,A -85,B 0,C 180,E1 -21913.094,E2 -21913.094} C_VEL
LIN {X 0,Y 192.49,Z 255.503,A -85,B 0,C 180,E1 -21916.904,E2 -21916.904} C_VEL
LIN {X 0,Y 192.551,Z 255.489,A -85,B 0,C 180,E1 -21921.648,E2 -21921.648} C_VEL
LIN {X 0,Y 192.596,Z 255.482,A -85,B 0,C 180,E1 -21926.813,E2 -21926.813} C_VEL
LIN {X 0,Y 192.66,Z 255.483,A -85,B 0,C 180,E1 -21931.691,E2 -21931.691} C_VEL
LIN {X 0,Y 192.705,Z 255.448,A -85,B 0,C 180,E1 -21936.348,E2 -21936.348} C_VEL
LIN {X 0,Y 192.731,Z 255.474,A -85,B 0,C 180,E1 -21941.457,E2 -21941.457} C_VEL
LIN {X 0,Y 192.771,Z 255.465,A -85,B 0,C 180,E1 -21945.214,E2 -21945.214} C_VEL
LIN {X 0,Y 193.019,Z 255.405,A -85,B 0,C 180,E1 -21949.51,E2 -21949.51} C_VEL
LIN {X 0,Y 193.003,Z 255.439,A -85,B 0,C 180,E1 -21953.728,E2 -21953.728} C_VEL
LIN {X 0,Y 193.263,Z 255.405,A -85,B 0,C 180,E1 -21957.916,E2 -21957.916} C_VEL
LIN {X 0,Y 193.442,Z 255.367,A -85,B 0,C 180,E1 -21960,E2 -21960} C_VEL
LIN {X 0,Y 192.977,Z 255.429,A -85,B 0,C 180,E1 -21964.177,E2 -21964.177} C_VEL
LIN {X 0,Y 193.078,Z 255.434,A -85,B 0,C 180,E1 -21968.372,E2 -21968.372} C_VEL
LIN {X 0,Y 193.009,Z 255.434,A -85,B 0,C 180,E1 -21970.538,E2 -21970.538} C_VEL
LIN {X 0,Y 192.756,Z 255.472,A -85,B 0,C 180,E1 -21976.959,E2 -21976.959} C_VEL
LIN {X 0,Y 192.635,Z 255.481,A -85,B 0,C 180,E1 -21981.397,E2 -21981.397} C_VEL
LIN {X 0,Y 192.663,Z 255.482,A -85,B 0,C 180,E1 -21984.225,E2 -21984.225} C_VEL
LIN {X 0,Y 192.649,Z 255.48,A -85,B 0,C 180,E1 -21988.892,E2 -21988.892} C_VEL
LIN {X 0,Y 192.598,Z 255.488,A -85,B 0,C 180,E1 -21993.186,E2 -21993.186} C_VEL
LIN {X 0,Y 192.55,Z 255.496,A -85,B 0,C 180,E1 -21998.352,E2 -21998.352} C_VEL
LIN {X 0,Y 192.488,Z 255.492,A -85,B 0,C 180,E1 -22003.096,E2 -22003.096} C_VEL
LIN {X 0,Y 192.551,Z 255.693,A -85,B 0,C 180,E1 -22007.204,E2 -22007.204} C_VEL
LIN {X 0,Y 193.96,Z 261.029,A -85,B 0,C 180,E1 -22010.149,E2 -22010.149} C_VEL
LIN {X 0,Y 201.826,Z 277.805,A -85,B 0,C 180,E1 -22012.392,E2 -22012.392} C_VEL
LIN {X 0,Y 209.42,Z 296.609,A -85,B 0,C 180,E1 -22014.47,E2 -22014.47} C_VEL
LIN {X 0,Y 210.845,Z 301.502,A -85,B 0,C 180,E1 -22014.898,E2 -22014.898} C_VEL
LIN {X 0,Y 212.85,Z 317.492,A -85,B 0,C 180,E1 -22015.854,E2 -22015.854} C_VEL
LIN {X 0,Y 212.222,Z 333.343,A -85,B 0,C 180,E1 -22016.398,E2 -22016.398} C_VEL
LIN {X 0,Y 211.309,Z 339.18,A -85,B 0,C 180,E1 -22016.498,E2 -22016.498} C_VEL
LIN {X 0,Y 205.234,Z 358.077,A -85,B 0,C 180,E1 -22016.368,E2 -22016.368} C_VEL
LIN {X 0,Y 204.469,Z 363.899,A -85,B 0,C 180,E1 -22016.508,E2 -22016.508} C_VEL
LIN {X 0,Y 203.394,Z 377.353,A -85,B 0,C 180,E1 -22017.177,E2 -22017.177} C_VEL
LIN {X 0,Y 201.644,Z 390.403,A -85,B 0,C 180,E1 -22018.187,E2 -22018.187} C_VEL
LIN {X 0,Y 199.448,Z 402.76,A -85,B 0,C 180,E1 -22019.567,E2 -22019.567} C_VEL
LIN {X 0,Y 197.108,Z 413.911,A -85,B 0,C 180,E1 -22021.227,E2 -22021.227} C_VEL
LIN {X 0,Y 194.673,Z 424.15,A -85,B 0,C 180,E1 -22023.175,E2 -22023.175} C_VEL
LIN {X 0,Y 191.871,Z 434.465,A -85,B 0,C 180,E1 -22025.665,E2 -22025.665} C_VEL
LIN {X 0,Y 189.65,Z 442.877,A -85,B 0,C 180,E1 -22028.249,E2 -22028.249} C_VEL
LIN {X 0,Y 187.672,Z 449.837,A -85,B 0,C 180,E1 -22030.873,E2 -22030.873} C_VEL
LIN {X 0,Y 185.756,Z 456.65,A -85,B 0,C 180,E1 -22034.08,E2 -22034.08} C_VEL
LIN {X 0,Y 184.255,Z 462.89,A -85,B 0,C 180,E1 -22037.891,E2 -22037.891} C_VEL
LIN {X 0,Y 183.505,Z 466.92,A -85,B 0,C 180,E1 -22041.188,E2 -22041.188} C_VEL
LIN {X 0,Y 183.21,Z 468.982,A -85,B 0,C 180,E1 -22043.392,E2 -22043.392} C_VEL
LIN {X 0,Y 183.042,Z 471.25,A -85,B 0,C 180,E1 -22046.646,E2 -22046.646} C_VEL
LIN {X 0,Y 183.186,Z 472.624,A -85,B 0,C 180,E1 -22050,E2 -22050} C_VEL
LIN {X 0,Y 183.053,Z 473.03,A -85,B 0,C 180,E1 -22053.414,E2 -22053.414} C_VEL
LIN {X 0,Y 183.212,Z 472.525,A -85,B 0,C 180,E1 -22056.609,E2 -22056.609} C_VEL
LIN {X 0,Y 183.512,Z 471.708,A -85,B 0,C 180,E1 -22058.812,E2 -22058.812} C_VEL
LIN {X 0,Y 184.785,Z 468.821,A -85,B 0,C 180,E1 -22063.191,E2 -22063.191} C_VEL
LIN {X 0,Y 186.333,Z 465.555,A -85,B 0,C 180,E1 -22066.432,E2 -22066.432} C_VEL
LIN {X 0,Y 188.622,Z 461.245,A -85,B 0,C 180,E1 -22069.593,E2 -22069.593} C_VEL
LIN {X 0,Y 191.836,Z 454.764,A -85,B 0,C 180,E1 -22073.193,E2 -22073.193} C_VEL
LIN {X 0,Y 195.103,Z 447.704,A -85,B 0,C 180,E1 -22076.185,E2 -22076.185} C_VEL
LIN {X 0,Y 198.979,Z 438.931,A -85,B 0,C 180,E1 -22079.056,E2 -22079.056} C_VEL
LIN {X 0,Y 203.112,Z 429.02,A -85,B 0,C 180,E1 -22081.557,E2 -22081.557} C_VEL
LIN {X 0,Y 206.725,Z 418.974,A -85,B 0,C 180,E1 -22083.535,E2 -22083.535} C_VEL
LIN {X 0,Y 210.198,Z 407.886,A -85,B 0,C 180,E1 -22085.223,E2 -22085.223} C_VEL
LIN {X 0,Y 213.356,Z 395.532,A -85,B 0,C 180,E1 -22086.658,E2 -22086.658} C_VEL
LIN {X 0,Y 215.873,Z 382.993,A -85,B 0,C 180,E1 -22087.694,E2 -22087.694} C_VEL
LIN {X 0,Y 217.721,Z 369.739,A -85,B 0,C 180,E1 -22088.434,E2 -22088.434} C_VEL
LIN {X 0,Y 219.67,Z 341.42,A -85,B 0,C 180,E1 -22089.399,E2 -22089.399} C_VEL
LIN {X 0,Y 220.906,Z 321.576,A -85,B 0,C 180,E1 -22090.046,E2 -22090.046} C_VEL
LIN {X 0,Y 220.335,Z 317.44,A -85,B 0,C 180,E1 -22090.405,E2 -22090.405} C_VEL
LIN {X 0,Y 215.619,Z 305.675,A -85,B 0,C 180,E1 -22092.377,E2 -22092.377} C_VEL
LIN {X 0,Y 210.701,Z 295.447,A -85,B 0,C 180,E1 -22094.525,E2 -22094.525} C_VEL
LIN {X 0,Y 205.321,Z 285.859,A -85,B 0,C 180,E1 -22097.074,E2 -22097.074} C_VEL
LIN {X 0,Y 201.736,Z 280.078,A -85,B 0,C 180,E1 -22098.911,E2 -22098.911} C_VEL
LIN {X 0,Y 198.907,Z 275.653,A -85,B 0,C 180,E1 -22100.506,E2 -22100.506} C_VEL
LIN {X 0,Y 195.274,Z 270.238,A -85,B 0,C 180,E1 -22102.733,E2 -22102.733} C_VEL
LIN {X 0,Y 191.979,Z 265.924,A -85,B 0,C 180,E1 -22104.95,E2 -22104.95} C_VEL
LIN {X 0,Y 190.994,Z 264.298,A -85,B 0,C 180,E1 -22105.705,E2 -22105.705} C_VEL
LIN {X 0,Y 187.065,Z 259.872,A -85,B 0,C 180,E1 -22108.897,E2 -22108.897} C_VEL
LIN {X 0,Y 185.819,Z 257.52,A -85,B 0,C 180,E1 -22110.269,E2 -22110.269} C_VEL
LIN {X 0,Y 185.587,Z 256.355,A -85,B 0,C 180,E1 -22112.055,E2 -22112.055} C_VEL
LIN {X 0,Y 185.589,Z 256.363,A -85,B 0,C 180,E1 -22115.383,E2 -22115.383} C_VEL
LIN {X 0,Y 185.676,Z 256.342,A -85,B 0,C 180,E1 -22121.133,E2 -22121.133} C_VEL
LIN {X 0,Y 185.725,Z 256.341,A -85,B 0,C 180,E1 -22124.64,E2 -22124.64} C_VEL
LIN {X 0,Y 185.925,Z 256.315,A -85,B 0,C 180,E1 -22129.359,E2 -22129.359} C_VEL
LIN {X 0,Y 185.961,Z 256.316,A -85,B 0,C 180,E1 -22133.49,E2 -22133.49} C_VEL
LIN {X 0,Y 186.208,Z 256.288,A -85,B 0,C 180,E1 -22137.837,E2 -22137.837} C_VEL
LIN {X 0,Y 186.405,Z 256.252,A -85,B 0,C 180,E1 -22140,E2 -22140} C_VEL
LIN {X 0,Y 185.951,Z 256.498,A -85,B 0,C 180,E1 -22145.286,E2 -22145.286} C_VEL
LIN {X 0,Y 186.632,Z 258.614,A -85,B 0,C 180,E1 -22146.08,E2 -22146.08} C_VEL
LIN {X 0,Y 188.541,Z 260.942,A -85,B 0,C 180,E1 -22147.766,E2 -22147.766} C_VEL
LIN {X 0,Y 190.731,Z 262.419,A -85,B 0,C 180,E1 -22149.403,E2 -22149.403} C_VEL
LIN {X 0,Y 192.296,Z 265.422,A -85,B 0,C 180,E1 -22150.643,E2 -22150.643} C_VEL
LIN {X 0,Y 194.934,Z 268.027,A -85,B 0,C 180,E1 -22152.361,E2 -22152.361} C_VEL
LIN {X 0,Y 197.283,Z 271.48,A -85,B 0,C 180,E1 -22153.848,E2 -22153.848} C_VEL
LIN {X 0,Y 198.928,Z 273.242,A -85,B 0,C 180,E1 -22154.776,E2 -22154.776} C_VEL
LIN {X 0,Y 202.749,Z 278.652,A -85,B 0,C 180,E1 -22156.872,E2 -22156.872} C_VEL
LIN {X 0,Y 206.113,Z 283.4,A -85,B 0,C 180,E1 -22158.528,E2 -22158.528} C_VEL
LIN {X 0,Y 211.286,Z 291.332,A -85,B 0,C 180,E1 -22160.888,E2 -22160.888} C_VEL
LIN {X 0,Y 216.689,Z 301.656,A -85,B 0,C 180,E1 -22163.18,E2 -22163.18} C_VEL
LIN {X 0,Y 221.289,Z 312.018,A -85,B 0,C 180,E1 -22165.035,E2 -22165.035} C_VEL
LIN {X 0,Y 221.109,Z 317.708,A -85,B 0,C 180,E1 -22165.268,E2 -22165.268} C_VEL
